# B&R Automation Studio project Parker_BMM_ST_V5_3147_V12 (part 22)

```c
				gPanelObj.idxKeyPicture[S$KEYMATRIX_F5] = STATE_SUB_PAGE;
					if(1 == EDGEPOS(gPanelObj.KeyMatric[S$KEYMATRIX_F5],KeyMatric[S$KEYMATRIX_F5]))
					{
					if(gPanelObj.PasswordLevel > 3)gPanelObj.SetPicture = PIC_OEM_SETTING_1;
				}
				if(gPanelObj.PasswordLevel <= 3)gPanelObj.idxKeyPicture[S$KEYMATRIX_F5] = STATE_INACTIVE;

					gPanelObj.idxKeyPicture[S$KEYMATRIX_F6] = STATE_SUB_PAGE;
					if(1 == EDGEPOS(gPanelObj.KeyMatric[S$KEYMATRIX_F6],KeyMatric[S$KEYMATRIX_F6]))
					{
					if(gPanelObj.PasswordLevel > 0)gPanelObj.SetPicture = PIC_PASSWORD_SET;
				}
				gPanelObj.idxKeyPicture[S$KEYMATRIX_F7] = STATE_SUB_PAGE;
					if(1 == EDGEPOS(gPanelObj.KeyMatric[S$KEYMATRIX_F7],KeyMatric[S$KEYMATRIX_F7]))
					{
					if(gPanelObj.PasswordLevel > 2)gPanelObj.SetPicture = PIC_PRESSURE_CALIBRATION ;
				}
				if(gPanelObj.PasswordLevel <= 2)gPanelObj.idxKeyPicture[S$KEYMATRIX_F7] = STATE_INACTIVE;
					//				gPanelObj.idxKeyPicture[S$KEYMATRIX_F7] = STATE_SUB_PAGE;
					//				if(1 == EDGEPOS(gPanelObj.KeyMatric[S$KEYMATRIX_F7],KeyMatric[S$KEYMATRIX_F7]))
					//				{
					//					if(0 == bLevel3CalibHide)
					//					{
					//						gPanelObj.SetPicture = PIC_MOLD_CALIBRATION;
					//					}
					//				}
					//				if(1 == bLevel3CalibHide)gPanelObj.idxKeyPicture[S$KEYMATRIX_F7] = STATE_INACTIVE;

					gPanelObj.idxKeyPicture[S$KEYMATRIX_F8] = STATE_SUB_PAGE;
					if(1 == EDGEPOS(gPanelObj.KeyMatric[S$KEYMATRIX_F8],KeyMatric[S$KEYMATRIX_F8]))
					{
					if(0 == bLevel3CalibHide)
					{
						if(ACTUATOR_ELECTRIC == gMachineFix.MoldR.Clamp.eActuatorType)
						{
							gPanelObj.SetPicture = PIC_CALIB_CLAMP_ENCODER;
						}
						else if(ACTUATOR_HYD == gMachineFix.MoldR.Clamp.eActuatorType )
						{
							gPanelObj.SetPicture = PIC_CALIB_CLAMP_LVDT;
						}

					}
				}
				if(1 == bLevel3CalibHide)gPanelObj.idxKeyPicture[S$KEYMATRIX_F8] = STATE_INACTIVE;

					//				gPanelObj.idxKeyPicture[S$KEYMATRIX_F7] = STATE_INACTIVE;
					//				gPanelObj.idxKeyPicture[S$KEYMATRIX_F8] = STATE_INACTIVE;

					gPanelObj.idxKeyPicture[S$KEYMATRIX_F9] = STATE_SUB_PAGE;
					if(1 == EDGEPOS(gPanelObj.KeyMatric[S$KEYMATRIX_F9],KeyMatric[S$KEYMATRIX_F9]))
					{
					if(gPanelObj.PasswordLevel > 3 && 1 == gTKcalib.Status)
					{
						gPanelObj.SetPicture = PIC_PROPORTION_VALVE;
					}
				}
				if(1 == bHidePropValvePage)gPanelObj.idxKeyPicture[S$KEYMATRIX_F9] = STATE_INACTIVE;

					gPanelObj.idxKeyPicture[S$KEYMATRIX_F10] = STATE_SUB_PAGE;
					if(1 == EDGEPOS(gPanelObj.KeyMatric[S$KEYMATRIX_F10],KeyMatric[S$KEYMATRIX_F10]))
					{
					gPanelObj.SetPicture = PIC_SCREEN_CALIBRATE;
				}

				gPanelObj.idxKeyPicture[S$KEYMATRIX_F11] = STATE_SUB_PAGE;
					if(1 == EDGEPOS(gPanelObj.KeyMatric[S$KEYMATRIX_F11],KeyMatric[S$KEYMATRIX_F11]))
					{
					if(gPanelObj.PasswordLevel > 2)gPanelObj.SetPicture = PIC_PV_LOG;
				}
				if(gPanelObj.PasswordLevel < 3)gPanelObj.idxKeyPicture[S$KEYMATRIX_F11] = STATE_INACTIVE;

					gPanelObj.idxKeyPicture[S$KEYMATRIX_F12] = STATE_SUB_PAGE;
					if(1 == EDGEPOS(gPanelObj.KeyMatric[S$KEYMATRIX_F12],KeyMatric[S$KEYMATRIX_F12]))
					{
					if(gPanelObj.PasswordLevel > 2)gPanelObj.SetPicture = PIC_LOG_INFO;
				}
				if(gPanelObj.PasswordLevel < 3)gPanelObj.idxKeyPicture[S$KEYMATRIX_F12] = STATE_INACTIVE;

					gPanelObj.idxKeyPicture[S$KEYMATRIX_F13] = STATE_SUB_PAGE;
					if(1 == EDGEPOS(gPanelObj.KeyMatric[S$KEYMATRIX_F13],KeyMatric[S$KEYMATRIX_F13]))
					{
					if(gPanelObj.PasswordLevel > 0)gPanelObj.SetPicture = PIC_INDUSTY_40;
				}
				if(gPanelObj.PasswordLevel < 1)gPanelObj.idxKeyPicture[S$KEYMATRIX_F13] = STATE_INACTIVE;

					gPanelObj.idxKeyPicture[S$KEYMATRIX_F14] = STATE_SUB_PAGE;
					if(1 == EDGEPOS(gPanelObj.KeyMatric[S$KEYMATRIX_F14],KeyMatric[S$KEYMATRIX_F14]))
					{
					if(gPanelObj.PasswordLevel > 0)gPanelObj.SetPicture = PIC_IP_CONFIG;
				}
				if(gPanelObj.PasswordLevel < 1)gPanelObj.idxKeyPicture[S$KEYMATRIX_F14] = STATE_INACTIVE;

					gPanelObj.idxKeyPicture[S$KEYMATRIX_F15] = STATE_SUB_PAGE;
					if(1 == EDGEPOS(gPanelObj.KeyMatric[S$KEYMATRIX_F15],KeyMatric[S$KEYMATRIX_F15]))
					{
					if(gPanelObj.PasswordLevel > 0)gPanelObj.SetPicture = PIC_VNC;
				}

				//						gPanelObj.idxKeyPicture[S$KEYMATRIX_F7] = STATE_INACTIVE;
				//            		gPanelObj.idxKeyPicture[S$KEYMATRIX_F8] = STATE_INACTIVE;
				//						gPanelObj.idxKeyPicture[S$KEYMATRIX_F8] = STATE_SUB_BUTTON;
				//						if(1 == EDGEPOS(gPanelObj.KeyMatric[S$KEYMATRIX_F8],KeyMatric[S$KEYMATRIX_F8]))
				//						{
				//						gMachineInfo.CycleTimes = 0;
				//						gCycleTimes             = 0;
				//						gMachineInfo.GoodBottles = 0;
				//					}

				//					gPanelObj.idxKeyPicture[S$KEYMATRIX_F9] = STATE_INACTIVE;
				//					gPanelObj.idxKeyPicture[S$KEYMATRIX_F10] = STATE_INACTIVE;
				//						gPanelObj.idxKeyPicture[S$KEYMATRIX_F10] = STATE_SUB_PAGE;
				//						if(1 == EDGEPOS(gPanelObj.KeyMatric[S$KEYMATRIX_F10],KeyMatric[S$KEYMATRIX_F10]))
				//						{
				//						gPanelObj.SetPicture = PIC_SCREEN_CALIBRATE;
				//					}
				//					gPanelObj.idxKeyPicture[S$KEYMATRIX_F11] = STATE_INACTIVE;
				//						gPanelObj.idxKeyPicture[S$KEYMATRIX_F12] = STATE_INACTIVE;
				//						gPanelObj.idxKeyPicture[S$KEYMATRIX_F13] = STATE_INACTIVE;
				//						gPanelObj.idxKeyPicture[S$KEYMATRIX_F14] = STATE_INACTIVE;
				//						gPanelObj.idxKeyPicture[S$KEYMATRIX_F15] = STATE_INACTIVE;

				gPanelObj.idxKeyPicture[S$KEYMATRIX_F16] = STATE_SUB_PAGE;
					if(1 == EDGEPOS(gPanelObj.KeyMatric[S$KEYMATRIX_F16],KeyMatric[S$KEYMATRIX_F16]))
					{
					gPanelObj.SetPicture = PIC_PASSWORD_LOGIN;
				}

				break;

			case PIC_PASSWORD_SET:
				//	case PIC_VALVE_DELAY:
			case PIC_PV_LOG:
				if(ChangePageDly > 0)
				{
					ChangePageDly--;
					break;
				}

				gPanelObj.idxKeyPicture[S$KEYMATRIX_F1] = STATE_SUB_PAGE;
				if(1 == EDGEPOS(gPanelObj.KeyMatric[S$KEYMATRIX_F1],KeyMatric[S$KEYMATRIX_F1]))
					{
					gPanelObj.SetPicture = PIC_OVERVIEW;
				}

				gPanelObj.idxKeyPicture[S$KEYMATRIX_F2] = STATE_SUB_PAGE;
					if(1 == EDGEPOS(gPanelObj.KeyMatric[S$KEYMATRIX_F2],KeyMatric[S$KEYMATRIX_F2]))
					{
					gPanelObj.SetPicture = gPanelObj.OldPicture;
				}

				gPanelObj.idxKeyPicture[S$KEYMATRIX_F3] = STATE_INACTIVE;
					gPanelObj.idxKeyPicture[S$KEYMATRIX_F4] = STATE_INACTIVE;
					gPanelObj.idxKeyPicture[S$KEYMATRIX_F5] = STATE_INACTIVE;

					gPanelObj.idxKeyPicture[S$KEYMATRIX_F6] = STATE_SUB_BUTTON;
					gPanelObj.idxKeyPicture[S$KEYMATRIX_F7] = STATE_SUB_BUTTON;

					gPanelObj.idxKeyPicture[S$KEYMATRIX_F8] = STATE_INACTIVE;
					gPanelObj.idxKeyPicture[S$KEYMATRIX_F9] = STATE_INACTIVE;
					gPanelObj.idxKeyPicture[S$KEYMATRIX_F10] = STATE_INACTIVE;
					gPanelObj.idxKeyPicture[S$KEYMATRIX_F11] = STATE_INACTIVE;
					gPanelObj.idxKeyPicture[S$KEYMATRIX_F12] = STATE_INACTIVE;
					gPanelObj.idxKeyPicture[S$KEYMATRIX_F13] = STATE_INACTIVE;
					gPanelObj.idxKeyPicture[S$KEYMATRIX_F14] = STATE_INACTIVE;
					gPanelObj.idxKeyPicture[S$KEYMATRIX_F15] = STATE_INACTIVE;
					gPanelObj.idxKeyPicture[S$KEYMATRIX_F16] = STATE_SUB_PAGE;
					if(1 == EDGEPOS(gPanelObj.KeyMatric[S$KEYMATRIX_F16],KeyMatric[S$KEYMATRIX_F16]))
					{
					gPanelObj.SetPicture = PIC_PASSWORD_LOGIN;
				}
				break;

			case PIC_SPC_CTRL:
			case PIC_SPC_1:
			case PIC_SPC_2:
				if(ChangePageDly > 0)
				{
					ChangePageDly--;
					break;
				}

				gPanelObj.idxKeyPicture[S$KEYMATRIX_F1] = STATE_SUB_PAGE;
					if(1 == EDGEPOS(gPanelObj.KeyMatric[S$KEYMATRIX_F1],KeyMatric[S$KEYMATRIX_F1]))
					{
					gPanelObj.SetPicture = PIC_OVERVIEW;
				}

				gPanelObj.idxKeyPicture[S$KEYMATRIX_F2] = STATE_SUB_PAGE;
					if(1 == EDGEPOS(gPanelObj.KeyMatric[S$KEYMATRIX_F2],KeyMatric[S$KEYMATRIX_F2]))
					{
					gPanelObj.SetPicture = gPanelObj.OldPicture;
				}

				gPanelObj.idxKeyPicture[S$KEYMATRIX_F3] = STATE_SUB_PAGE;
					if(1 == EDGEPOS(gPanelObj.KeyMatric[S$KEYMATRIX_F3],KeyMatric[S$KEYMATRIX_F3]))
					{
					gPanelObj.SetPicture = PIC_SPC_CTRL;
				}

				if(PIC_SPC_CTRL == gPanelObj.GetPicture)gPanelObj.idxKeyPicture[S$KEYMATRIX_F3]=STATE_ACTIVE;

					gPanelObj.idxKeyPicture[S$KEYMATRIX_F4] = STATE_SUB_PAGE;
					if(1 == EDGEPOS(gPanelObj.KeyMatric[S$KEYMATRIX_F4],KeyMatric[S$KEYMATRIX_F4]))
					{
					gPanelObj.SetPicture = PIC_SPC_1;
				}

				if(PIC_SPC_1 == gPanelObj.GetPicture)gPanelObj.idxKeyPicture[S$KEYMATRIX_F4]=STATE_ACTIVE;

					gPanelObj.idxKeyPicture[S$KEYMATRIX_F5] = STATE_SUB_PAGE;
					if(1 == EDGEPOS(gPanelObj.KeyMatric[S$KEYMATRIX_F5],KeyMatric[S$KEYMATRIX_F5]))
					{
					gPanelObj.SetPicture = PIC_SPC_2;
				}

				if(PIC_SPC_2 == gPanelObj.GetPicture)gPanelObj.idxKeyPicture[S$KEYMATRIX_F5]=STATE_ACTIVE;

					gPanelObj.idxKeyPicture[S$KEYMATRIX_F6] = STATE_INACTIVE;

					if(gPanelObj.GetPicture != PIC_SPC_CTRL)
				{
					gPanelObj.idxKeyPicture[S$KEYMATRIX_F7] = STATE_SUB_BUTTON;
						gPanelObj.idxKeyPicture[S$KEYMATRIX_F8] = STATE_SUB_BUTTON;
						}
				else
				{
					gPanelObj.idxKeyPicture[S$KEYMATRIX_F7] = STATE_INACTIVE;
						gPanelObj.idxKeyPicture[S$KEYMATRIX_F8] = STATE_INACTIVE;
						}

				gPanelObj.idxKeyPicture[S$KEYMATRIX_F9] = STATE_INACTIVE;
					gPanelObj.idxKeyPicture[S$KEYMATRIX_F10] = STATE_INACTIVE;
					gPanelObj.idxKeyPicture[S$KEYMATRIX_F11] = STATE_INACTIVE;
					gPanelObj.idxKeyPicture[S$KEYMATRIX_F12] = STATE_INACTIVE;
					gPanelObj.idxKeyPicture[S$KEYMATRIX_F13] = STATE_INACTIVE;
					gPanelObj.idxKeyPicture[S$KEYMATRIX_F14] = STATE_INACTIVE;
					gPanelObj.idxKeyPicture[S$KEYMATRIX_F15] = STATE_INACTIVE;
					gPanelObj.idxKeyPicture[S$KEYMATRIX_F16] = STATE_SUB_PAGE;
					if(1 == EDGEPOS(gPanelObj.KeyMatric[S$KEYMATRIX_F16],KeyMatric[S$KEYMATRIX_F16]))
					{
					gPanelObj.SetPicture = PIC_PASSWORD_LOGIN;
				}
				break;

			case PIC_HIGH_PASSWORD:
				if(ChangePageDly > 0)
				{
					ChangePageDly--;
					break;
				}

				gPanelObj.idxKeyPicture[S$KEYMATRIX_F1] = STATE_SUB_PAGE;
					if(1 == EDGEPOS(gPanelObj.KeyMatric[S$KEYMATRIX_F1],KeyMatric[S$KEYMATRIX_F1]))
					{
					gPanelObj.SetPicture = PIC_OVERVIEW;
				}

				gPanelObj.idxKeyPicture[S$KEYMATRIX_F2] = STATE_SUB_PAGE;
					if(1 == EDGEPOS(gPanelObj.KeyMatric[S$KEYMATRIX_F2],KeyMatric[S$KEYMATRIX_F2]))
					{
					gPanelObj.SetPicture = gPanelObj.OldPicture;
				}

				gPanelObj.idxKeyPicture[S$KEYMATRIX_F3] = STATE_INACTIVE;

					gPanelObj.idxKeyPicture[S$KEYMATRIX_F4] = STATE_INACTIVE;
					if(1 == EDGEPOS(gPanelObj.KeyMatric[S$KEYMATRIX_F4],KeyMatric[S$KEYMATRIX_F4]))
					{
					if(PIC_HIGH_PASSWORD == gPanelObj.GetPicture)
					{
						gPwd.Option[0] = !gPwd.Option[0];
						gPwd.wSavePassword = 1;
					}
				}
				if(gPanelObj.GetPicture == PIC_HIGH_PASSWORD)gPanelObj.idxKeyPicture[S$KEYMATRIX_F4] = STATE_SUB_BUTTON;

					gPanelObj.idxKeyPicture[S$KEYMATRIX_F5] = STATE_INACTIVE;
					if(1 == EDGEPOS(gPanelObj.KeyMatric[S$KEYMATRIX_F5],KeyMatric[S$KEYMATRIX_F5]))
					{
					if(PIC_HIGH_PASSWORD == gPanelObj.GetPicture)
					{
						gPwd.Option[1] = !gPwd.Option[1];
						gPwd.wSavePassword = 1;
					}
				}
				if(gPanelObj.GetPicture == PIC_HIGH_PASSWORD)gPanelObj.idxKeyPicture[S$KEYMATRIX_F5] = STATE_SUB_BUTTON;

					gPanelObj.idxKeyPicture[S$KEYMATRIX_F6] = STATE_INACTIVE;
					if(1 == EDGEPOS(gPanelObj.KeyMatric[S$KEYMATRIX_F6],KeyMatric[S$KEYMATRIX_F6]))
					{
					if(PIC_HIGH_PASSWORD == gPanelObj.GetPicture)
					{
						gPwd.Option[2] = !gPwd.Option[2];
						gPwd.wSavePassword = 1;
					}
				}
				if(gPanelObj.GetPicture == PIC_HIGH_PASSWORD)gPanelObj.idxKeyPicture[S$KEYMATRIX_F6] = STATE_SUB_BUTTON;

					gPanelObj.idxKeyPicture[S$KEYMATRIX_F7] = STATE_INACTIVE;

					gPanelObj.idxKeyPicture[S$KEYMATRIX_F8] = STATE_INACTIVE;
					if(1 == EDGEPOS(gPanelObj.KeyMatric[S$KEYMATRIX_F8],KeyMatric[S$KEYMATRIX_F8]))
					{
					if(PIC_HIGH_PASSWORD == gPanelObj.GetPicture)
					{
						gMachineStopDays = 0;

						gPwd.OK_3 = 0;
						gPwd.OK_2 = 0;
						gPwd.OK_1 = 0;

						gPwd.wSavePassword = 1;
					}
				}
				if(gPanelObj.GetPicture == PIC_HIGH_PASSWORD)gPanelObj.idxKeyPicture[S$KEYMATRIX_F8] = STATE_SUB_BUTTON;

					gPanelObj.idxKeyPicture[S$KEYMATRIX_F9] = STATE_INACTIVE;
					gPanelObj.idxKeyPicture[S$KEYMATRIX_F10] = STATE_INACTIVE;
					gPanelObj.idxKeyPicture[S$KEYMATRIX_F11] = STATE_INACTIVE;
					gPanelObj.idxKeyPicture[S$KEYMATRIX_F12] = STATE_INACTIVE;
					gPanelObj.idxKeyPicture[S$KEYMATRIX_F13] = STATE_INACTIVE;
					if(gPanelObj.GetPicture == PIC_INDUSTY_40)gPanelObj.idxKeyPicture[S$KEYMATRIX_F13] = STATE_ACTIVE;
					gPanelObj.idxKeyPicture[S$KEYMATRIX_F14] = STATE_INACTIVE;
					gPanelObj.idxKeyPicture[S$KEYMATRIX_F15] = STATE_INACTIVE;
					gPanelObj.idxKeyPicture[S$KEYMATRIX_F16] = STATE_SUB_PAGE;
					if(1 == EDGEPOS(gPanelObj.KeyMatric[S$KEYMATRIX_F16],KeyMatric[S$KEYMATRIX_F16]))
					{
					gPanelObj.SetPicture = PIC_PASSWORD_LOGIN;
				}
				break;

			case PIC_INIT_SET:
				if(ChangePageDly > 0)
				{
					ChangePageDly--;
					break;
				}

				gPanelObj.idxKeyPicture[S$KEYMATRIX_F1] = STATE_SUB_PAGE;
					if(1 == EDGEPOS(gPanelObj.KeyMatric[S$KEYMATRIX_F1],KeyMatric[S$KEYMATRIX_F1]))
					{
					gPanelObj.SetPicture = PIC_OVERVIEW;
				}

				gPanelObj.idxKeyPicture[S$KEYMATRIX_F2] = STATE_SUB_PAGE;
					if(1 == EDGEPOS(gPanelObj.KeyMatric[S$KEYMATRIX_F2],KeyMatric[S$KEYMATRIX_F2]))
					{
					gPanelObj.SetPicture = gPanelObj.OldPicture;
				}

				gPanelObj.idxKeyPicture[S$KEYMATRIX_F3] = STATE_ACTIVE;
					if(1 == EDGEPOS(gPanelObj.KeyMatric[S$KEYMATRIX_F3],KeyMatric[S$KEYMATRIX_F3]))
					{
					gPanelObj.SetPicture = PIC_THICK_START;
				}
				gPanelObj.idxKeyPicture[S$KEYMATRIX_F4] = STATE_INACTIVE;
					gPanelObj.idxKeyPicture[S$KEYMATRIX_F5] = STATE_INACTIVE;
					gPanelObj.idxKeyPicture[S$KEYMATRIX_F6] = STATE_INACTIVE;
					gPanelObj.idxKeyPicture[S$KEYMATRIX_F7] = STATE_INACTIVE;
					gPanelObj.idxKeyPicture[S$KEYMATRIX_F8] = STATE_INACTIVE;
					gPanelObj.idxKeyPicture[S$KEYMATRIX_F9] = STATE_INACTIVE;
					gPanelObj.idxKeyPicture[S$KEYMATRIX_F10] = STATE_INACTIVE;
					gPanelObj.idxKeyPicture[S$KEYMATRIX_F11] = STATE_INACTIVE;

					if(1 == EDGEPOS(gPanelObj.KeyMatric[S$KEYMATRIX_F12],KeyMatric[S$KEYMATRIX_F12]))
					{
					gPanelObj.SetPicture = PIC_THICK_DIVER;
				}
				//					gPanelObj.idxKeyPicture[S$KEYMATRIX_F6] = STATE_SUB_BUTTON;
				//					if(1 == EDGEPOS(gPanelObj.KeyMatric[S$KEYMATRIX_F6],KeyMatric[S$KEYMATRIX_F6]))
				//					{
				//					gThickProf.FunOption.bLengthUnit = !gThickProf.FunOption.bLengthUnit;
				//					gRecipeOperate.OnceSave = 1;
				//				}
				//
				//				gPanelObj.idxKeyPicture[S$KEYMATRIX_F7] = STATE_SUB_BUTTON;
				//					if(1 == EDGEPOS(gPanelObj.KeyMatric[S$KEYMATRIX_F7],KeyMatric[S$KEYMATRIX_F7]))
				//					{
				//					gThickProf.FunOption.IsTraceInEdit = !gThickProf.FunOption.IsTraceInEdit;
				//					gRecipeOperate.OnceSave = 1;
				//				}
				//
				//				gPanelObj.idxKeyPicture[S$KEYMATRIX_F8] = STATE_SUB_BUTTON;
				//					if(1 == EDGEPOS(gPanelObj.KeyMatric[S$KEYMATRIX_F8],KeyMatric[S$KEYMATRIX_F8]))
				//					{
				//					gThickProf.FunOption.Is100_300 = !gThickProf.FunOption.Is100_300;
				//					gRecipeOperate.OnceSave = 1;
				//				}
				//
				//				gPanelObj.idxKeyPicture[S$KEYMATRIX_F9] = STATE_SUB_BUTTON;
				//					if(1 == EDGEPOS(gPanelObj.KeyMatric[S$KEYMATRIX_F9],KeyMatric[S$KEYMATRIX_F9]))
				//					{
				//					gThickProf.FunOption.IsZeroDn = !gThickProf.FunOption.IsZeroDn;
				//					gRecipeOperate.OnceSave = 1;
				//				}
				//
				//				gPanelObj.idxKeyPicture[S$KEYMATRIX_F10] = STATE_SUB_BUTTON;
				//					if(1 == EDGEPOS(gPanelObj.KeyMatric[S$KEYMATRIX_F10],KeyMatric[S$KEYMATRIX_F10]))
				//					{
				//					gThickProf.FunOption.SealMode = !gThickProf.FunOption.SealMode;
				//					gRecipeOperate.OnceSave = 1;
				//				}
				//
				//				gPanelObj.idxKeyPicture[S$KEYMATRIX_F11] = STATE_INACTIVE;
				//
				//					gPanelObj.idxKeyPicture[S$KEYMATRIX_F12] = STATE_SUB_BUTTON;
				//					if(1 == EDGEPOS(gPanelObj.KeyMatric[S$KEYMATRIX_F12],KeyMatric[S$KEYMATRIX_F12]))
				//					{
				//					gThickProf.FunOption.Servo = !gThickProf.FunOption.Servo;
				//					gRecipeOperate.OnceSave = 1;
				//				}

				gPanelObj.idxKeyPicture[S$KEYMATRIX_F13] = STATE_SUB_PAGE;
					if(1 == EDGENEG(gPanelObj.KeyMatric[S$KEYMATRIX_F13],KeyMatric[S$KEYMATRIX_F13]))
					{
					//	if(gPanelObj.PasswordLevel > 2 &&  1 == gTKcalib.Status)
					if(gPanelObj.PasswordLevel > 2 &&  0 == gTKauto.Status)

					{
						gPanelObj.SetPicture = PIC_INIT_SET  ;
						OldSet    = gThickProf.ShareSet;
						OldFunSet = gThickProf.FunOption;
					}
				}
				//	if(1 == bThickCalibHide)gPanelObj.idxKeyPicture[S$KEYMATRIX_F13] = STATE_INACTIVE;
				if(1 == gTKauto.Status)gPanelObj.idxKeyPicture[S$KEYMATRIX_F13] = STATE_INACTIVE;

					gPanelObj.idxKeyPicture[S$KEYMATRIX_F14] = STATE_SUB_PAGE;
					if(1 == EDGENEG(gPanelObj.KeyMatric[S$KEYMATRIX_F14],KeyMatric[S$KEYMATRIX_F14]))
					{
					//	if(gPanelObj.PasswordLevel > 2 &&  1 == gTKcalib.Status)
					if(gPanelObj.PasswordLevel > 2 &&  0 == gTKauto.Status)
					{
						gPanelObj.SetPicture = PIC_GAP_CALIBRATE;
						OldSet    = gThickProf.ShareSet;
						OldFunSet = gThickProf.FunOption;
					}
				}
				//if(1 == bThickCalibHide)gPanelObj.idxKeyPicture[S$KEYMATRIX_F14] = STATE_INACTIVE;
				if(1 == gTKauto.Status)gPanelObj.idxKeyPicture[S$KEYMATRIX_F14] = STATE_INACTIVE;
					gPanelObj.idxKeyPicture[S$KEYMATRIX_F15] = STATE_INACTIVE;
					gPanelObj.idxKeyPicture[S$KEYMATRIX_F16] = STATE_SUB_PAGE;
					if(1 == EDGEPOS(gPanelObj.KeyMatric[S$KEYMATRIX_F16],KeyMatric[S$KEYMATRIX_F16]))
					{
					gPanelObj.SetPicture = PIC_PASSWORD_LOGIN;
				}

				if(gThickProf.ShareSet.StartFlow > 998)gThickProf.ShareSet.StartFlow = 998;
				if(gThickProf.ShareSet.SealFlow  > 998)gThickProf.ShareSet.SealFlow  = 998;
				if(gThickProf.ShareSet.ThickFlow > 998)gThickProf.ShareSet.ThickFlow = 998;

				if(gThickProf.ShareSet.StartFlow < 100)gThickProf.ShareSet.StartFlow = 100;
				if(gThickProf.ShareSet.SealFlow  < 100)gThickProf.ShareSet.SealFlow  = 100;
				if(gThickProf.ShareSet.ThickFlow < 100)gThickProf.ShareSet.ThickFlow = 100;
				break;

			case PIC_GAP_CALIBRATE:
				if(ChangePageDly > 0)
				{
					ChangePageDly--;
					break;
				}

				gPanelObj.idxKeyPicture[S$KEYMATRIX_F1] = STATE_SUB_PAGE;
					if(1 == EDGEPOS(gPanelObj.KeyMatric[S$KEYMATRIX_F1],KeyMatric[S$KEYMATRIX_F1]))
					{
					gPanelObj.SetPicture = PIC_OVERVIEW;
				}

				gPanelObj.idxKeyPicture[S$KEYMATRIX_F2] = STATE_SUB_PAGE;
					if(1 == EDGEPOS(gPanelObj.KeyMatric[S$KEYMATRIX_F2],KeyMatric[S$KEYMATRIX_F2]))
					{
					gPanelObj.SetPicture = gPanelObj.OldPicture;
				}

				gPanelObj.idxKeyPicture[S$KEYMATRIX_F3] = STATE_ACTIVE;
					if(1 == EDGEPOS(gPanelObj.KeyMatric[S$KEYMATRIX_F3],KeyMatric[S$KEYMATRIX_F3]))
					{
					gPanelObj.SetPicture = PIC_THICK_START;
				}
				gPanelObj.idxKeyPicture[S$KEYMATRIX_F4]  = STATE_INACTIVE;

					if(gMachineFix.Parison.eActuatorType == ACTUATOR_ELECTRIC)
				{
					//Electric

					if (gPanelObj.GetPicture ==PIC_GAP_CALIBRATE )
					{
						gPanelObj.idxKeyPicture[S$KEYMATRIX_F5] = STATE_SUB_BUTTON;
							if(1 == EDGEPOS(gPanelObj.KeyMatric[S$KEYMATRIX_F5],KeyMatric[S$KEYMATRIX_F5]))
							{
							if(1 == gMachineInfo.Calib)
							{
								gThickIO.Step = STEP_THICK_CALIB_DOWN;
							}
						}

						if(1 == EDGENEG(gPanelObj.KeyMatric[S$KEYMATRIX_F5],keyF5N))
							{
							if(1 == gMachineInfo.Calib)
							{
								gThickIO.Step = STEP_THICK_STOP;
							}
						}

						gPanelObj.idxKeyPicture[S$KEYMATRIX_F6] = STATE_SUB_BUTTON;
							if(1 == EDGEPOS(gPanelObj.KeyMatric[S$KEYMATRIX_F6],KeyMatric[S$KEYMATRIX_F6]))
							{
							if(1 == gMachineInfo.Calib)
							{
								gThickIO.Step = STEP_THICK_CALIB_UP;
							}
						}

						if(1 == EDGENEG(gPanelObj.KeyMatric[S$KEYMATRIX_F6],keyF6N))
							{
							if(1 == gMachineInfo.Calib)
							{
								gThickIO.Step = STEP_THICK_STOP;
							}
						}
						gPanelObj.idxKeyPicture[S$KEYMATRIX_F7] = STATE_SUB_BUTTON;
							if(1 == EDGEPOS(gPanelObj.KeyMatric[S$KEYMATRIX_F7],KeyMatric[S$KEYMATRIX_F7]))
							{
							if(1 == gMachineInfo.Calib)
							{
								gThickFix.ecMin = gThickIO.ecAs;
								gRecipeOperate.OnceSave = 1;
							}
						}

						gPanelObj.idxKeyPicture[S$KEYMATRIX_F8] = STATE_SUB_BUTTON;
							if(1 == EDGEPOS(gPanelObj.KeyMatric[S$KEYMATRIX_F8],KeyMatric[S$KEYMATRIX_F8]))
							{
							if(1 == gMachineInfo.Calib)
							{
								gThickFix.ecMax = gThickIO.ecAs;
								gRecipeOperate.OnceSave = 1;
							}
						}
					}

					gPanelObj.idxKeyPicture[S$KEYMATRIX_F9]  = STATE_INACTIVE;
						gPanelObj.idxKeyPicture[S$KEYMATRIX_F10] = STATE_INACTIVE;
						gPanelObj.idxKeyPicture[S$KEYMATRIX_F11] = STATE_INACTIVE;

						gPanelObj.idxKeyPicture[S$KEYMATRIX_F12] = STATE_SUB_PAGE;
						if(1 == EDGEPOS(gPanelObj.KeyMatric[S$KEYMATRIX_F12],KeyMatric[S$KEYMATRIX_F12]))
						{
						gPanelObj.SetPicture = PIC_THICK_DIVER;
					}

				}
				else if(gMachineFix.Parison.eActuatorType == ACTUATOR_HYD)
				{
					//Hydraulic

					gPanelObj.idxKeyPicture[S$KEYMATRIX_F5] = STATE_SUB_BUTTON;
						gPanelObj.idxKeyPicture[S$KEYMATRIX_F6] = STATE_SUB_BUTTON;
						gPanelObj.idxKeyPicture[S$KEYMATRIX_F7] = STATE_SUB_BUTTON;
						if(1 == gPanelObj.KeyMatric[S$KEYMATRIX_F7])
						{
						cntF7 = cntF7 + 1;
					}
					else
					{
						cntF7 = 0;
					}
					if(50 == cntF7)
					{
						if(gServoLinear.Current > 0 && gServoLinear.Current < 32767)
						{
							gServoLinear.ZeroPos     = gServoLinear.Current;
							gRecipeOperate.OnceSave = 1;
						}
					}

					gPanelObj.idxKeyPicture[S$KEYMATRIX_F8] = STATE_SUB_BUTTON;
						if(1 == gPanelObj.KeyMatric[S$KEYMATRIX_F8])
						{
						cntF8 = cntF8 + 1;
					}
					else
					{
						cntF8 = 0;
					}

					if(50 == cntF8)
					{
						if(gServoLinear.Current > 0 && gServoLinear.Current < 32767)
						{
							if(gServoLinear.Current > gServoLinear.ZeroPos)
							{
								gServoLinear.MaxPos      = gServoLinear.Current;
								gRecipeOperate.OnceSave = 1;
							}
						}
					}

					// auto calibration
					if(1 == gThickProf.FunOption.IsAutoCalibrate)
					{
						gPanelObj.idxKeyPicture[S$KEYMATRIX_F11] = STATE_SUB_BUTTON;
							bHideParisonAutoCalib = 0;

						if(1 == gPanelObj.KeyMatric[S$KEYMATRIX_F5] || 1 == gPanelObj.KeyMatric[S$KEYMATRIX_F6] ||
							1 == gPanelObj.KeyMatric[S$KEYMATRIX_F7] || 1 == gPanelObj.KeyMatric[S$KEYMATRIX_F8])
							{
							gImply.ParisonCalibNotManual = 1;
						}
					}
					else
					{
						gPanelObj.idxKeyPicture[S$KEYMATRIX_F11] = STATE_INACTIVE;
							bHideParisonAutoCalib = 1;
					}

					gPanelObj.idxKeyPicture[S$KEYMATRIX_F9]  = STATE_INACTIVE;
						gPanelObj.idxKeyPicture[S$KEYMATRIX_F10] = STATE_INACTIVE;

						gPanelObj.idxKeyPicture[S$KEYMATRIX_F12] = STATE_INACTIVE;

						}

				/*-------------------F13----------------------*/
				gPanelObj.idxKeyPicture[S$KEYMATRIX_F13] = STATE_SUB_PAGE;
					if(1 == EDGENEG(gPanelObj.KeyMatric[S$KEYMATRIX_F13],KeyMatric[S$KEYMATRIX_F13]))
					{
					//	if(gPanelObj.PasswordLevel > 2 &&  1 == gTKcalib.Status)
					if(gPanelObj.PasswordLevel > 2 &&  0 == gTKauto.Status)

					{
						gPanelObj.SetPicture = PIC_INIT_SET  ;
						OldSet    = gThickProf.ShareSet;
						OldFunSet = gThickProf.FunOption;
					}
				}

				if(1 == gTKauto.Status)gPanelObj.idxKeyPicture[S$KEYMATRIX_F13] = STATE_INACTIVE;

					/*-------------------F14----------------------*/
					gPanelObj.idxKeyPicture[S$KEYMATRIX_F14] = STATE_SUB_PAGE;
					if(1 == EDGENEG(gPanelObj.KeyMatric[S$KEYMATRIX_F14],KeyMatric[S$KEYMATRIX_F14]))
					{
					//	if(gPanelObj.PasswordLevel > 2 &&  1 == gTKcalib.Status)
					if(gPanelObj.PasswordLevel > 2 &&  0 == gTKauto.Status)
					{
						gPanelObj.SetPicture = PIC_GAP_CALIBRATE;
						OldSet    = gThickProf.ShareSet;
						OldFunSet = gThickProf.FunOption;
					}
				}
				//if(1 == bThickCalibHide)gPanelObj.idxKeyPicture[S$KEYMATRIX_F14] = STATE_INACTIVE;
				if(1 == gTKauto.Status)gPanelObj.idxKeyPicture[S$KEYMATRIX_F14] = STATE_INACTIVE;
					if(1 == EDGEPOS(gPanelObj.KeyMatric[S$KEYMATRIX_F15],KeyMatric[S$KEYMATRIX_F15]))
					{
					gPanelObj.SetPicture = PIC_GAP_CALIBRATE_HELP;
				}
				gPanelObj.idxKeyPicture[S$KEYMATRIX_F16] = STATE_SUB_PAGE;
					if(1 == EDGEPOS(gPanelObj.KeyMatric[S$KEYMATRIX_F16],KeyMatric[S$KEYMATRIX_F16]))
					{
					gPanelObj.SetPicture = PIC_PASSWORD_LOGIN;
				}
				break;

			case PIC_GAP_CALIBRATE_HELP:
				if(ChangePageDly > 0)
				{
					ChangePageDly--;
					break;
				}

				gPanelObj.idxKeyPicture[S$KEYMATRIX_F1] = STATE_SUB_PAGE;
					if(1 == EDGEPOS(gPanelObj.KeyMatric[S$KEYMATRIX_F1],KeyMatric[S$KEYMATRIX_F1]))
					{
					gPanelObj.SetPicture = PIC_GAP_CALIBRATE;
				}

				gPanelObj.idxKeyPicture[S$KEYMATRIX_F2] = STATE_INACTIVE;
					gPanelObj.idxKeyPicture[S$KEYMATRIX_F3] = STATE_INACTIVE;
					gPanelObj.idxKeyPicture[S$KEYMATRIX_F4] = STATE_INACTIVE;
					gPanelObj.idxKeyPicture[S$KEYMATRIX_F5] = STATE_INACTIVE;
					gPanelObj.idxKeyPicture[S$KEYMATRIX_F6] = STATE_INACTIVE;
					gPanelObj.idxKeyPicture[S$KEYMATRIX_F7] = STATE_INACTIVE;
					gPanelObj.idxKeyPicture[S$KEYMATRIX_F8] = STATE_INACTIVE;
					gPanelObj.idxKeyPicture[S$KEYMATRIX_F9] = STATE_INACTIVE;
					gPanelObj.idxKeyPicture[S$KEYMATRIX_F10] = STATE_INACTIVE;
					gPanelObj.idxKeyPicture[S$KEYMATRIX_F11] = STATE_INACTIVE;
					gPanelObj.idxKeyPicture[S$KEYMATRIX_F12] = STATE_INACTIVE;
					gPanelObj.idxKeyPicture[S$KEYMATRIX_F13] = STATE_INACTIVE;
					gPanelObj.idxKeyPicture[S$KEYMATRIX_F14] = STATE_INACTIVE;
					gPanelObj.idxKeyPicture[S$KEYMATRIX_F15] = STATE_INACTIVE;
					gPanelObj.idxKeyPicture[S$KEYMATRIX_F16] = STATE_SUB_PAGE;
					if(1 == EDGEPOS(gPanelObj.KeyMatric[S$KEYMATRIX_F16],KeyMatric[S$KEYMATRIX_F16]))
					{
					gPanelObj.SetPicture = PIC_PASSWORD_LOGIN;
				}
				break;

			case PIC_DEFAULT_SET:
				if(ChangePageDly > 0)
				{
					ChangePageDly--;
					break;
				}

				gPanelObj.idxKeyPicture[S$KEYMATRIX_F1] = STATE_SUB_PAGE;
					if(1 == EDGEPOS(gPanelObj.KeyMatric[S$KEYMATRIX_F1],KeyMatric[S$KEYMATRIX_F1]))
					{
					gPanelObj.SetPicture = PIC_OVERVIEW;
				}

				gPanelObj.idxKeyPicture[S$KEYMATRIX_F2] = STATE_SUB_PAGE;
					if(1 == EDGEPOS(gPanelObj.KeyMatric[S$KEYMATRIX_F2],KeyMatric[S$KEYMATRIX_F2]))
					{
					gPanelObj.SetPicture = gPanelObj.OldPicture;
				}

				gPanelObj.idxKeyPicture[S$KEYMATRIX_F3] = STATE_SUB_PAGE;
					if(1 == EDGEPOS(gPanelObj.KeyMatric[S$KEYMATRIX_F3],KeyMatric[S$KEYMATRIX_F3]))
					{
					gPanelObj.SetPicture = PIC_GAP_CALIBRATE;
				}

				gPanelObj.idxKeyPicture[S$KEYMATRIX_F4] = STATE_INACTIVE;
					gPanelObj.idxKeyPicture[S$KEYMATRIX_F5] = STATE_INACTIVE;
					gPanelObj.idxKeyPicture[S$KEYMATRIX_F6] = STATE_INACTIVE;
					gPanelObj.idxKeyPicture[S$KEYMATRIX_F7] = STATE_INACTIVE;
					gPanelObj.idxKeyPicture[S$KEYMATRIX_F8] = STATE_INACTIVE;
					gPanelObj.idxKeyPicture[S$KEYMATRIX_F9] = STATE_INACTIVE;

					gPanelObj.idxKeyPicture[S$KEYMATRIX_F10] = STATE_INACTIVE;
					gPanelObj.idxKeyPicture[S$KEYMATRIX_F11] = STATE_INACTIVE;
					gPanelObj.idxKeyPicture[S$KEYMATRIX_F12] = STATE_INACTIVE;
					gPanelObj.idxKeyPicture[S$KEYMATRIX_F13] = STATE_INACTIVE;
					gPanelObj.idxKeyPicture[S$KEYMATRIX_F14] = STATE_INACTIVE;
					gPanelObj.idxKeyPicture[S$KEYMATRIX_F15] = STATE_INACTIVE;
					gPanelObj.idxKeyPicture[S$KEYMATRIX_F16] = STATE_SUB_PAGE;
					if(1 == EDGEPOS(gPanelObj.KeyMatric[S$KEYMATRIX_F16],KeyMatric[S$KEYMATRIX_F16]))
					{
					gPanelObj.SetPicture = PIC_PASSWORD_LOGIN;
				}
				break;

			case PIC_CALIB_CLAMP_ENCODER:
			case PIC_CALIB_CARRIAGE_ENCODER:
			case PIC_CALIB_BLOWPIN_ENCODER:
			case PIC_CALIB_OTHER_ENCODER:
			case PIC_CALIB_ROBOT_ENCODER:
			case PIC_CALIB_CLAMP_LVDT:
			case PIC_CALIB_CARRIAGE_LVDT:
			case PIC_CALIB_BLOWPIN_LVDT:

				if(ChangePageDly > 0)
				{
					ChangePageDly--;
					break;
				}

				gPanelObj.idxKeyPicture[S$KEYMATRIX_F1] = STATE_SUB_PAGE;
					if(1 == EDGEPOS(gPanelObj.KeyMatric[S$KEYMATRIX_F1],KeyMatric[S$KEYMATRIX_F1]))
					{
					gPanelObj.SetPicture = PIC_OVERVIEW;
				}

				gPanelObj.idxKeyPicture[S$KEYMATRIX_F2] = STATE_SUB_PAGE;
					if(1 == EDGEPOS(gPanelObj.KeyMatric[S$KEYMATRIX_F2],KeyMatric[S$KEYMATRIX_F2]))
					{
					gPanelObj.SetPicture = gPanelObj.OldPicture;
				}

				gPanelObj.idxKeyPicture[S$KEYMATRIX_F3] = STATE_SUB_PAGE;
					if(1 == EDGEPOS(gPanelObj.KeyMatric[S$KEYMATRIX_F3],KeyMatric[S$KEYMATRIX_F3]))
					{
					gPanelObj.SetPicture = PIC_CALIB_CLAMP_ENCODER;
				}
				if( 1 == bHideClampActuatorElectic )gPanelObj.idxKeyPicture[S$KEYMATRIX_F3] = STATE_INACTIVE;

					gPanelObj.idxKeyPicture[S$KEYMATRIX_F4] = STATE_SUB_PAGE;
					if(1 == EDGEPOS(gPanelObj.KeyMatric[S$KEYMATRIX_F4],KeyMatric[S$KEYMATRIX_F4]))
					{
					gPanelObj.SetPicture = PIC_CALIB_CARRIAGE_ENCODER;

				}
				if( 1 == bHideCarriageActuatorElectic )gPanelObj.idxKeyPicture[S$KEYMATRIX_F4] = STATE_INACTIVE;

					gPanelObj.idxKeyPicture[S$KEYMATRIX_F5] = STATE_SUB_PAGE;
					if(1 == EDGEPOS(gPanelObj.KeyMatric[S$KEYMATRIX_F5],KeyMatric[S$KEYMATRIX_F5]))
					{
					gPanelObj.SetPicture = PIC_CALIB_BLOWPIN_ENCODER;
				}
				if( 1 == bHideBlowPinActuatorElectic)gPanelObj.idxKeyPicture[S$KEYMATRIX_F5] = STATE_INACTIVE;

					gPanelObj.idxKeyPicture[S$KEYMATRIX_F6] = STATE_SUB_PAGE;
					if(1 == EDGEPOS(gPanelObj.KeyMatric[S$KEYMATRIX_F6],KeyMatric[S$KEYMATRIX_F6]))
					{
					if( 0 == bHideClampActuatorHyd_LVDT)gPanelObj.SetPicture = PIC_CALIB_CLAMP_LVDT;
				}
				if( 1 == bHideClampActuatorHyd_LVDT)gPanelObj.idxKeyPicture[S$KEYMATRIX_F6] = STATE_INACTIVE;

					gPanelObj.idxKeyPicture[S$KEYMATRIX_F7] = STATE_SUB_PAGE;
					if(1 == EDGEPOS(gPanelObj.KeyMatric[S$KEYMATRIX_F7],KeyMatric[S$KEYMATRIX_F7]))
					{
					if( 0 == bHideCarriageActuatorHyd_LVDT)gPanelObj.SetPicture = PIC_CALIB_CARRIAGE_LVDT;
				}
				if( 1 == bHideCarriageActuatorHyd_LVDT)gPanelObj.idxKeyPicture[S$KEYMATRIX_F7] = STATE_INACTIVE;

					gPanelObj.idxKeyPicture[S$KEYMATRIX_F8] = STATE_SUB_PAGE;
					if(1 == EDGEPOS(gPanelObj.KeyMatric[S$KEYMATRIX_F8],KeyMatric[S$KEYMATRIX_F8]))
					{
					if( 0 == bHideBlowPinActuatorHyd_LVDT)gPanelObj.SetPicture = PIC_CALIB_BLOWPIN_LVDT;
				}
				if( 1 == bHideBlowPinActuatorHyd_LVDT)gPanelObj.idxKeyPicture[S$KEYMATRIX_F8] = STATE_INACTIVE;

					gPanelObj.idxKeyPicture[S$KEYMATRIX_F9] = STATE_SUB_PAGE;
					if(1 == EDGEPOS(gPanelObj.KeyMatric[S$KEYMATRIX_F9],KeyMatric[S$KEYMATRIX_F9]))
					{
					gPanelObj.SetPicture = PIC_CALIB_OTHER_ENCODER;
				}
				if( 1 == bHideExtrLiftActuatorElectric)gPanelObj.idxKeyPicture[S$KEYMATRIX_F9] = STATE_INACTIVE;

					gPanelObj.idxKeyPicture[S$KEYMATRIX_F10] = STATE_SUB_PAGE;
					if(1 == EDGEPOS(gPanelObj.KeyMatric[S$KEYMATRIX_F10],KeyMatric[S$KEYMATRIX_F10]))
					{
					gPanelObj.SetPicture = PIC_CALIB_ROBOT_ENCODER;
				}
				if( 1 == bHideRobotTransferActuatorElec)gPanelObj.idxKeyPicture[S$KEYMATRIX_F10] = STATE_INACTIVE;

					gPanelObj.idxKeyPicture[S$KEYMATRIX_F11] = STATE_INACTIVE;
					gPanelObj.idxKeyPicture[S$KEYMATRIX_F12] = STATE_INACTIVE;

					/*----Reset Calibrate Function---------*/
					/* check commands */
					if (((bCmdResetClampR) || (bCmdResetClampL) || (bCmdResetBlowPinR) || (bCmdResetBlowPinL) || (bCmdResetCarriageR) || (bCmdResetCarriageL)|| (bCmdResetBlowPin2R) || (bCmdResetBlowPin2L) || (bCmdResetExtrLift) )&& (gPanelObj.PasswordLevel > 3))
				{
					uHideDiagResetCalib = 0;
				}

				/*Dialog Pop up contorl*/

				if(0 == uHideDiagResetCalib)
				{
					if(bConfirmReset)
					{
						if(bCmdResetClampR)
						{
							gMachineFix.MoldR.Clamp.Zero = 0;
							gMachineFix.MoldR.Clamp.Max = 0;
							gRecipeOperate.OnceSave = 1;
							bCmdResetClampR = 0;
						}
						else if(bCmdResetClampL)
						{
							gMachineFix.MoldL.Clamp.Zero = 0;
							gMachineFix.MoldL.Clamp.Max = 0;
							gRecipeOperate.OnceSave = 1;
							bCmdResetClampL = 0;
						}
						else if(bCmdResetBlowPinR)
						{
							gMachineFix.MoldR.BlowPin.Zero = 0;
							gMachineFix.MoldR.BlowPin.Max = 0;
							gRecipeOperate.OnceSave = 1;
							bCmdResetBlowPinR = 0;
						}
						else if(bCmdResetBlowPinL)
						{
							gMachineFix.MoldL.BlowPin.Zero = 0;
							gMachineFix.MoldL.BlowPin.Max = 0;
							gRecipeOperate.OnceSave = 1;
							bCmdResetBlowPinL = 0;
						}
						else if(bCmdResetCarriageR)
						{
							gMachineFix.MoldR.Carriage.Zero = 0;
							gMachineFix.MoldR.Carriage.Max = 0;
							gRecipeOperate.OnceSave = 1;
							bCmdResetCarriageR = 0;
						}
						else if(bCmdResetCarriageL)
						{
							gMachineFix.MoldL.Carriage.Zero = 0;
							gMachineFix.MoldL.Carriage.Max = 0;
							gRecipeOperate.OnceSave = 1;
							bCmdResetCarriageL = 0;
						}
						else if(bCmdResetBlowPin2R)
						{
							gMachineFix.MoldR.BlowPin2.Zero = 0;
							gMachineFix.MoldR.BlowPin2.Max = 0;
							gRecipeOperate.OnceSave = 1;
							bCmdResetBlowPin2R = 0;
						}
						else if(bCmdResetBlowPin2L)
						{
							gMachineFix.MoldL.BlowPin2.Zero = 0;
							gMachineFix.MoldL.BlowPin2.Max = 0;
							gRecipeOperate.OnceSave = 1;
							bCmdResetBlowPin2L = 0;
						}
						else if(bCmdResetExtrLift)
						{
							gMachineFix.ExtrLift.Zero = 0;
							gMachineFix.ExtrLift.Max = 0;
							gRecipeOperate.OnceSave = 1;
							bCmdResetExtrLift = 0;
						}
						uHideDiagResetCalib = 1;
						bCancelReset = 	0;
						bConfirmReset = 0;
					}
					else if (bCancelReset)
					{
						bCancelReset = 	0;
						bConfirmReset = 0;
						uHideDiagResetCalib = 1;
						bCmdResetClampR = 0;
						bCmdResetClampL = 0;
						bCmdResetBlowPinR = 0;
						bCmdResetBlowPinL = 0;
						bCmdResetBlowPin2R = 0;
						bCmdResetBlowPin2L = 0;
						bCmdResetCarriageR = 0;
						bCmdResetCarriageL = 0;
						bCmdResetExtrLift  =0;
					}
				}
				else
				{
					bCancelReset = 	0;
					bConfirmReset = 0;
					bCmdResetClampR = 0;
					bCmdResetClampL = 0;
					bCmdResetBlowPinR = 0;
					bCmdResetBlowPinL = 0;
					bCmdResetCarriageR = 0;
					bCmdResetCarriageL = 0;
					bCmdResetExtrLift  =0;
				}

				/*-------------------Calibration Confirm----------------------*/
				for(i=0;i<sizeof(CalibList)/2;i++)
				{
					CalibList[i] = 0;
				}

				CalibList[IndexCalib] = 1;

				gPanelObj.idxKeyPicture[S$KEYMATRIX_F13] = STATE_SUB_BUTTON;
					if(1 == gPanelObj.KeyMatric[S$KEYMATRIX_F13] && 1 == gTKcalib.Status)
					{
					cntF13 = cntF13 + 1;
				}
				else
				{
					cntF13 = 0;
				}

				if(cntF13 > 20)
				{
					if(1 == gMachineInfo.Calib && PIC_CALIB_CLAMP_ENCODER == gPanelObj.GetPicture )	/* 调校模式  */
					{
						switch(IndexCalib)
						{
							case 0:
								gMachineFix.MoldL.Clamp.Zero = LMold.Clamp.As;
								gRecipeOperate.OnceSave= 1;

								break;
							case 1:
								gMachineFix.MoldR.Clamp.Zero = RMold.Clamp.As;
								gRecipeOperate.OnceSave = 1;

								break;
							case 2:

								break;
							case 3:

								break;
							case 4:
								gMachineFix.MoldL.Clamp.Max = LMold.Clamp.As;
								gRecipeOperate.OnceSave = 1;

								break;

							case 5:
								gMachineFix.MoldR.Clamp.Max = RMold.Clamp.As;
								gRecipeOperate.OnceSave = 1;

								break;

							case 6:

								break;
							case 7:

								break;

						}/* switch(IndexCalib) */
					}/* if(1 == gMachineInfo.Calib)*/
					else if(1 == gMachineInfo.Calib && PIC_CALIB_CARRIAGE_ENCODER == gPanelObj.GetPicture)
					{
						switch(IndexCalib)
						{
							case 0:
								if(1 == LMold.TransDIn.CarriageFwLimit)
								{
									gMachineFix.MoldL.Carriage.Zero = LMold.Carriage.As;
									gRecipeOperate.OnceSave = 1;
								}
								else
								{
									gImply.LCarriageFw = 1;
								}
								break;
							case 1:
								if(1 == RMold.TransDIn.CarriageFwLimit)
								{
									gMachineFix.MoldR.Carriage.Zero = RMold.Carriage.As;
									gRecipeOperate.OnceSave = 1;
								}
								else
								{
									gImply.RCarriageFw = 1;
								}
								break;

							case 2:

								break;
							case 3:

								break;
							case 4:
								if(1 == LMold.TransDIn.CarriageBwLimit)
								{
									gMachineFix.MoldL.Carriage.Max = LMold.Carriage.As;
									gRecipeOperate.OnceSave = 1;
								}
								else
								{
									gImply.LCarriageBw = 1;
								}
								break;

							case 5:
								if(1 == RMold.TransDIn.CarriageBwLimit)
								{
									gMachineFix.MoldR.Carriage.Max = RMold.Carriage.As;
									gRecipeOperate.OnceSave = 1;
								}
								else
								{
									gImply.RCarriageBw = 1;
								}
								break;

							case 6:

								break;
							case 7:

								break;

						}/* switch(IndexCalib) */
					}
					else if(1 == gMachineInfo.Calib && PIC_CALIB_BLOWPIN_ENCODER == gPanelObj.GetPicture)
					{
						switch(IndexCalib)
						{
							case 0:
								if(1 == LMold.TransDIn.BlowPin2UpLimit)
								{
									gMachineFix.MoldL.BlowPin2.Zero = LMold.BlowPin2.As;
									gRecipeOperate.OnceSave = 1;
								}
								else
								{
									gImply.LPin2Up = 1;
								}
								break;
							case 1:
								if(1 == LMold.TransDIn.BlowPinUpLimit)
								{
									gMachineFix.MoldL.BlowPin.Zero = LMold.BlowPin.As;
									gRecipeOperate.OnceSave = 1;
								}
								else
								{
									gImply.LPinUp = 1;
								}
								break;

							case 2:
								if(1 == RMold.TransDIn.BlowPin2UpLimit)
								{
									gMachineFix.MoldR.BlowPin2.Zero = RMold.BlowPin2.As;
									gRecipeOperate.OnceSave = 1;
								}
								else
								{
									gImply.RPin2Up = 1;
								}
								break;
							case 3:
								if(1 == RMold.TransDIn.BlowPinUpLimit)
								{
									gMachineFix.MoldR.BlowPin.Zero = RMold.BlowPin.As;
									gRecipeOperate.OnceSave = 1;
								}
								else
								{
									gImply.RPinUp = 1;
								}
								break;
							case 4:
								gMachineFix.MoldL.BlowPin2.Max = LMold.BlowPin2.As;
								gRecipeOperate.OnceSave= 1;

								break;
							case 5:
								gMachineFix.MoldL.BlowPin.Max = LMold.BlowPin.As;
								gRecipeOperate.OnceSave = 1;

								break;

							case 6:
								gMachineFix.MoldR.BlowPin2.Max = RMold.BlowPin2.As;
								gRecipeOperate.OnceSave = 1;

								break;
							case 7:
								gMachineFix.MoldR.BlowPin.Max = RMold.BlowPin.As;
								gRecipeOperate.OnceSave = 1;

								break;

						}/* switch(IndexCalib) */
					}
					else if(1 == gMachineInfo.Calib && PIC_CALIB_OTHER_ENCODER == gPanelObj.GetPicture)
					{
						switch(IndexCalib)
						{
							case 0:

								break;
							case 1:
								if(1 == RMold.TransDIn.ExtruderLiftDnLimit)
								{
									gMachineFix.ExtrLift.Zero = RMold.ExtrLift.As;
									gRecipeOperate.OnceSave = 1;
								}
								else
								{
									gImply.ExtrLiftDn = 1;
								}

								break;

							case 2:

								break;
							case 3:

								break;
							case 4:

								break;
							case 5:
								//								if(1 == RMold.TransDIn.ExtruderLiftUpLimit)
								//								{
								gMachineFix.ExtrLift.Max = RMold.ExtrLift.As;
								gRecipeOperate.OnceSave = 1;
								//								}
								//								else
								//								{
								//									gImply.ExtrLiftUp = 1;
								//								}

								break;

							case 6:

								break;
							case 7:

								break;

						}/* switch(IndexCalib) */
					}
					else if(1 == gMachineInfo.Calib && PIC_CALIB_CLAMP_LVDT == gPanelObj.GetPicture)
					{
						switch(IndexCalib)
						{
							case 0:
								gMachineFix.MoldL.Clamp.Zero = LMold.Clamp.As;
								gRecipeOperate.OnceSave= 1;

								break;
							case 1:
								gMachineFix.MoldR.Clamp.Zero = RMold.Clamp.As;
								gRecipeOperate.OnceSave = 1;

								break;
							case 2:

								break;

							case 3:

								break;
							case 4:
								gMachineFix.MoldL.Clamp.Max = LMold.Clamp.As;
								gRecipeOperate.OnceSave = 1;

								break;
							case 5:
								gMachineFix.MoldR.Clamp.Max = RMold.Clamp.As;
								gRecipeOperate.OnceSave = 1;

								break;
							case 6:

								break;
							case 7:

								break;

						}/* switch(IndexCalib) */
					}
					else if(1 == gMachineInfo.Calib && PIC_CALIB_CARRIAGE_LVDT == gPanelObj.GetPicture)
					{
						switch(IndexCalib)
						{
							case 0:
								gMachineFix.MoldL.Carriage.Zero = LMold.Carriage.As;
								gRecipeOperate.OnceSave= 1;

								break;
							case 1:
								gMachineFix.MoldR.Carriage.Zero = RMold.Carriage.As;
								gRecipeOperate.OnceSave = 1;

								break;
							case 2:

								break;
							case 3:

								break;
							case 4:
								gMachineFix.MoldL.Carriage.Max = LMold.Carriage.As;
								gRecipeOperate.OnceSave = 1;

								break;
							case 5:
								gMachineFix.MoldR.Carriage.Max = RMold.Carriage.As;
								gRecipeOperate.OnceSave = 1;

								break;
							case 6:

								break;
							case 7:

								break;

						}/* switch(IndexCalib) */
					}
					else if(1 == gMachineInfo.Calib && PIC_CALIB_BLOWPIN_LVDT == gPanelObj.GetPicture)
					{
						switch(IndexCalib)
						{
							case 0:
								gMachineFix.MoldL.BlowPin.Zero = LMold.BlowPin.As;
								gRecipeOperate.OnceSave= 1;

								break;
							case 1:
								gMachineFix.MoldR.BlowPin.Zero = RMold.BlowPin.As;
								gRecipeOperate.OnceSave = 1;
								break;

							case 2:

								break;
							case 3:

								break;
							case 4:
								gMachineFix.MoldL.BlowPin.Max = LMold.BlowPin.As;
								gRecipeOperate.OnceSave = 1;

								break;

							case 5:
								gMachineFix.MoldR.BlowPin.Max = RMold.BlowPin.As;
								gRecipeOperate.OnceSave = 1;

								break;

							case 6:

								break;
							case 7:

								break;

						}/* switch(IndexCalib) */
					}
					else
					{
						gImply.CalMode = !gMachineInfo.Calib;
					}

				}/* if(1 == EDGEPOS(gPanelObj.KeyMatric[S$KEY_F13],KeyMatric[S$KEY_F13])) */

				// Robot Calib
				if(PIC_CALIB_ROBOT_ENCODER == gPanelObj.GetPicture)
				{
					if(1 == bRRobotHorZero)
					{
						cntRRobotHorZero++;
					}
					else
					{
						RMold.Robot.Transfer.Home = 0;
						cntRRobotHorZero =0;
					}

					if(1 == bRRobotVerZero)
					{
						RMold.Robot.UpDn.Home = 0;
						cntRRobotVerZero++;
					}
					else
					{
						cntRRobotVerZero =0;
					}

					if(1 == bLRobotHorZero)
					{
						cntLRobotHorZero++;
					}
					else
					{
						LMold.Robot.Transfer.Home = 0;
						cntLRobotHorZero =0;
					}

					if(1 == bLRobotVerZero)
					{
						cntLRobotVerZero++;
					}
					else
					{
						LMold.Robot.UpDn.Home =0;
						cntLRobotVerZero =0;
					}

					if(1 == gMachineInfo.Calib)	/* clibration mode  */
					{
						if(cntRRobotHorZero > 20)
						{
							if(1 == gMachineIn.RMold.RobotBwLimit)
							{
								gMachineFix.MoldR.RobotTransfer.sHome = RMold.Robot.Transfer.ecAs;
							}
							else
							{
								gImply.RRobotBw = 1;
							}
						}

						if(cntRRobotVerZero > 20)
						{
							if(1 == gMachineIn.RMold.RobotUpLimit)
							{
								gMachineFix.MoldR.RobotUpDn.sHome = RMold.Robot.UpDn.ecAs;
							}
							else
							{
								gImply.RRobotUp = 1;
							}
						}

						if(cntLRobotHorZero > 20)
						{
							if(1 == gMachineIn.LMold.RobotBwLimit)
							{
								gMachineFix.MoldL.RobotTransfer.sHome = LMold.Robot.Transfer.ecAs;
							}
							else
							{
								gImply.LRobotBw = 1;
							}
						}

						if(cntLRobotVerZero > 20)
						{
							if(1 == gMachineIn.LMold.RobotUpLimit)
							{
								gMachineFix.MoldL.RobotUpDn.sHome = LMold.Robot.UpDn.ecAs;
							}
							else
							{
								gImply.LRobotUp = 1;
							}
						}
					}
				}

				gPanelObj.idxKeyPicture[S$KEYMATRIX_F14] = STATE_INACTIVE;
					gPanelObj.idxKeyPicture[S$KEYMATRIX_F15] = STATE_INACTIVE;
					gPanelObj.idxKeyPicture[S$KEYMATRIX_F16] = STATE_SUB_PAGE;

					if(1 == EDGEPOS(gPanelObj.KeyMatric[S$KEYMATRIX_F16],KeyMatric[S$KEYMATRIX_F16]))
					{
					gPanelObj.SetPicture = PIC_PASSWORD_LOGIN;
				}
				break;

			case PIC_SCREEN_CALIBRATE:
				if(ChangePageDly > 0)
				{
					ChangePageDly--;
					break;
				}

				gPanelObj.idxKeyPicture[S$KEYMATRIX_F1] = STATE_SUB_PAGE;
					if(1 == EDGEPOS(gPanelObj.KeyMatric[S$KEYMATRIX_F1],KeyMatric[S$KEYMATRIX_F1]))
					{
					gPanelObj.SetPicture = PIC_OVERVIEW;
				}

				gPanelObj.idxKeyPicture[S$KEYMATRIX_F2] = STATE_SUB_PAGE;
					if(1 == EDGEPOS(gPanelObj.KeyMatric[S$KEYMATRIX_F2],KeyMatric[S$KEYMATRIX_F2]))
					{
					gPanelObj.SetPicture = gPanelObj.OldPicture;
				}

				gPanelObj.idxKeyPicture[S$KEYMATRIX_F3] = STATE_INACTIVE;
					gPanelObj.idxKeyPicture[S$KEYMATRIX_F4] = STATE_INACTIVE;
					gPanelObj.idxKeyPicture[S$KEYMATRIX_F5] = STATE_INACTIVE;
					gPanelObj.idxKeyPicture[S$KEYMATRIX_F6] = STATE_INACTIVE;
					gPanelObj.idxKeyPicture[S$KEYMATRIX_F7] = STATE_INACTIVE;
					gPanelObj.idxKeyPicture[S$KEYMATRIX_F8] = STATE_SUB_BUTTON;

					if(1 == EDGEPOS(gPanelObj.KeyMatric[S$KEYMATRIX_F8],KeyMatric[S$KEYMATRIX_F8]))
					{
					gPanelObj.vcHandle = VA_Setup(1, gPanelObj.VisualName);

					if (gPanelObj.vcHandle != 0)
					{
						if (!VA_Saccess(1, gPanelObj.vcHandle))
						{
							VA_StartTouchCal (1,gPanelObj.vcHandle);
							VA_Srelease(1, gPanelObj.vcHandle);
						}
					}
				}
				gPanelObj.idxKeyPicture[S$KEYMATRIX_F9] = STATE_INACTIVE;
					gPanelObj.idxKeyPicture[S$KEYMATRIX_F10] = STATE_INACTIVE;
					gPanelObj.idxKeyPicture[S$KEYMATRIX_F11] = STATE_INACTIVE;
					gPanelObj.idxKeyPicture[S$KEYMATRIX_F12] = STATE_INACTIVE;
					gPanelObj.idxKeyPicture[S$KEYMATRIX_F13] = STATE_INACTIVE;
					gPanelObj.idxKeyPicture[S$KEYMATRIX_F14] = STATE_INACTIVE;
					gPanelObj.idxKeyPicture[S$KEYMATRIX_F15] = STATE_INACTIVE;

					gPanelObj.idxKeyPicture[S$KEYMATRIX_F16] = STATE_SUB_PAGE;
					if(1 == EDGEPOS(gPanelObj.KeyMatric[S$KEYMATRIX_F16],KeyMatric[S$KEYMATRIX_F16]))
					{
					gPanelObj.SetPicture = PIC_PASSWORD_LOGIN;
				}
				if(ready == 0)
				{
					VC_HANDLE = VA_Setup(1 , gPanelObj.VisualName);

					if(VC_HANDLE != 0)ready = 1;
				}

				if(1 == ready)
				{
					if (!VA_Saccess(1,VC_HANDLE))
					{
						VA_GetTouchAction (1,VC_HANDLE,0,(UDINT)(&touch));
						VA_Ellipse (1,VC_HANDLE,touch.x,touch.y,2,2,0,0);
						VA_Srelease(1,VC_HANDLE);
					}
				}
				break;

			/*2018.8.3 Albert add new page for fast setting*/
			case PIC_FAST_SETTING:
				if(ChangePageDly > 0)
				{
					ChangePageDly--;
					break;
				}

				/*-----------F1---------*/
				gPanelObj.idxKeyPicture[S$KEYMATRIX_F1] = STATE_SUB_PAGE;
					if(1 == EDGEPOS(gPanelObj.KeyMatric[S$KEYMATRIX_F1],KeyMatric[S$KEYMATRIX_F1]))
					{
					gPanelObj.SetPicture = PIC_OVERVIEW;
				}
				/*-----------F2---------*/
				gPanelObj.idxKeyPicture[S$KEYMATRIX_F2] = STATE_SUB_PAGE;
					if(1 == EDGEPOS(gPanelObj.KeyMatric[S$KEYMATRIX_F2],KeyMatric[S$KEYMATRIX_F2]))
					{
					gPanelObj.SetPicture = gPanelObj.OldPicture;
				}
				/*-----------F3---------*/
				gPanelObj.idxKeyPicture[S$KEYMATRIX_F3] = STATE_SUB_PAGE;
					if(1 == bHideLeftStation)gPanelObj.idxKeyPicture[S$KEYMATRIX_F3] = STATE_INACTIVE;
					if(1 == EDGEPOS(gPanelObj.KeyMatric[S$KEYMATRIX_F3],KeyMatric[S$KEYMATRIX_F3]))
					{
					if(0 == bHideLeftStation)gPanelObj.SetPicture = PIC_CLAMP_L;
				}
				if(gPanelObj.GetPicture == PIC_CLAMP_L)gPanelObj.idxKeyPicture[S$KEYMATRIX_F3] = STATE_ACTIVE;

					/*-----------F4---------*/
					gPanelObj.idxKeyPicture[S$KEYMATRIX_F4] = STATE_SUB_PAGE;
					if(1 == EDGEPOS(gPanelObj.KeyMatric[S$KEYMATRIX_F4],KeyMatric[S$KEYMATRIX_F4]))
					{
					gPanelObj.SetPicture = PIC_CLAMP_R;
				}
				if(gPanelObj.GetPicture == PIC_CLAMP_R)gPanelObj.idxKeyPicture[S$KEYMATRIX_F4] = STATE_ACTIVE;

					/*-------------F5---------*/
					gPanelObj.idxKeyPicture[S$KEYMATRIX_F5] = STATE_SUB_PAGE;
					if(1 == bHideLeftStation)gPanelObj.idxKeyPicture[S$KEYMATRIX_F5] = STATE_INACTIVE;
					if(1 == EDGEPOS(gPanelObj.KeyMatric[S$KEYMATRIX_F5],KeyMatric[S$KEYMATRIX_F5]))
					{
					if(0 == bHideLeftStation)gPanelObj.SetPicture = PIC_TRANSPORT_L;
				}
				if(gPanelObj.GetPicture == PIC_TRANSPORT_L)gPanelObj.idxKeyPicture[S$KEYMATRIX_F5] = STATE_ACTIVE;

					/*------------F6-----------*/
					gPanelObj.idxKeyPicture[S$KEYMATRIX_F6] = STATE_SUB_PAGE;
					if(1 == EDGEPOS(gPanelObj.KeyMatric[S$KEYMATRIX_F6],KeyMatric[S$KEYMATRIX_F6]))
					{
					gPanelObj.SetPicture = PIC_TRANSPORT_R;
				}
				if(gPanelObj.GetPicture == PIC_TRANSPORT_R)gPanelObj.idxKeyPicture[S$KEYMATRIX_F6] = STATE_ACTIVE;

					/*------------F7-----------*/
					gPanelObj.idxKeyPicture[S$KEYMATRIX_F7] = STATE_SUB_PAGE;
					if(1 == bHideLeftStation)gPanelObj.idxKeyPicture[S$KEYMATRIX_F7] = STATE_INACTIVE;
					if(1 == EDGEPOS(gPanelObj.KeyMatric[S$KEYMATRIX_F7],KeyMatric[S$KEYMATRIX_F7]))
					{
					if(0 == bHideLeftStation)gPanelObj.SetPicture = PIC_BLOW_PIN_L;
				}
				if(gPanelObj.GetPicture == PIC_BLOW_PIN_L)gPanelObj.idxKeyPicture[S$KEYMATRIX_F7] = STATE_ACTIVE;

					/*-----------F8------------*/
					gPanelObj.idxKeyPicture[S$KEYMATRIX_F8] = STATE_SUB_PAGE;
					if(1 == EDGEPOS(gPanelObj.KeyMatric[S$KEYMATRIX_F8],KeyMatric[S$KEYMATRIX_F8]))
					{
					gPanelObj.SetPicture = PIC_BLOW_PIN_R;
				}
				if(gPanelObj.GetPicture == PIC_BLOW_PIN_R)gPanelObj.idxKeyPicture[S$KEYMATRIX_F8] = STATE_ACTIVE;

					/*----------F9-------------*/

					gPanelObj.idxKeyPicture[S$KEYMATRIX_F9] = STATE_SUB_PAGE;
					if(1 == EDGEPOS(gPanelObj.KeyMatric[S$KEYMATRIX_F9],KeyMatric[S$KEYMATRIX_F9]))
					{
					gPanelObj.SetPicture = PIC_DEFLASH;
				}
				if(gPanelObj.GetPicture == PIC_DEFLASH)gPanelObj.idxKeyPicture[S$KEYMATRIX_F9] = STATE_ACTIVE;

					/*----------F10-------------*/
					gPanelObj.idxKeyPicture[S$KEYMATRIX_F10] = STATE_INACTIVE;
					//						if(1 == EDGEPOS(gPanelObj.KeyMatric[S$KEYMATRIX_F10],KeyMatric[S$KEYMATRIX_F10]))
					//						{
					//						gPanelObj.SetPicture = PIC_BOTTOM_DEFLASH;
					//					}
					//					if(gPanelObj.GetPicture == PIC_BOTTOM_DEFLASH)gPanelObj.idxKeyPicture[S$KEYMATRIX_F10] = STATE_ACTIVE;

					gPanelObj.idxKeyPicture[S$KEYMATRIX_F11] = STATE_INACTIVE;
					//						if(1 == EDGEPOS(gPanelObj.KeyMatric[S$KEYMATRIX_F11],KeyMatric[S$KEYMATRIX_F11]))
					//						{
					//						gPanelObj.SetPicture = PIC_IO_DI_1;
					//					}

					gPanelObj.idxKeyPicture[S$KEYMATRIX_F12] = STATE_SUB_PAGE;
					if(1 == EDGEPOS(gPanelObj.KeyMatric[S$KEYMATRIX_F12],KeyMatric[S$KEYMATRIX_F12]))
					{
					gPanelObj.SetPicture = PIC_ALARM_CURRENT;
				}

				gPanelObj.idxKeyPicture[S$KEYMATRIX_F13] = STATE_SUB_PAGE;
					if(1 == EDGEPOS(gPanelObj.KeyMatric[S$KEYMATRIX_F13],KeyMatric[S$KEYMATRIX_F13]))
					{
					gPanelObj.SetPicture = PIC_AUTO_STEP;
				}

				gPanelObj.idxKeyPicture[S$KEYMATRIX_F14] = STATE_SUB_PAGE;
					if(1 == EDGEPOS(gPanelObj.KeyMatric[S$KEYMATRIX_F14],KeyMatric[S$KEYMATRIX_F14]))
					{
					gPanelObj.SetPicture = PIC_AUTO_START;
				}

				gPanelObj.idxKeyPicture[S$KEYMATRIX_F15] = STATE_SUB_PAGE;
					if(1 == EDGEPOS(gPanelObj.KeyMatric[S$KEYMATRIX_F15],KeyMatric[S$KEYMATRIX_F15]))
					{
					gPanelObj.SetPicture = PIC_SPC_CTRL;
				}

				gPanelObj.idxKeyPicture[S$KEYMATRIX_F16] = STATE_SUB_PAGE;
					if(1 == EDGEPOS(gPanelObj.KeyMatric[S$KEYMATRIX_F16],KeyMatric[S$KEYMATRIX_F16]))
					{
					gPanelObj.SetPicture = PIC_PASSWORD_LOGIN;
				}

				if(1 == EDGEPOS(gPanelObj.KeyMatric[S$KEYMATRIX_UP],KeyMatric[S$KEYMATRIX_UP]))
					{
					gPanelObj.SetLanguage = 1;
				}

				if(1 == EDGEPOS(gPanelObj.KeyMatric[S$KEYMATRIX_DOWN],KeyMatric[S$KEYMATRIX_DOWN]))
					{
					gPanelObj.SetLanguage = 0;
				}

				if(1 == EDGEPOS(gPanelObj.KeyMatric[S$KEYMATRIX_ESC],KeyMatric[S$KEYMATRIX_ESC]))
					{
					gPwd.PwdLevel = 0;
					gPanelObj.SetPicture = PIC_INIT;
				}

				//					/*Albert Machine Option*/
				//					for(i=0;i<OptionDis.Count;i++)
				//					{
				//						if(1 == HotSpot[i])
				//						{
				//							HotSpot[i]  = 0;
				//							if(0 == OptionDis.pHideSource[i])
				//							{
				//								OptionDis.Current = i;
				//								OptionDis.pSource[OptionDis.Current] = !OptionDis.pSource[OptionDis.Current];
				//								gRecipeOperate.DataSave = 1;
				//							}
				//						}
				//						OptionDis.Obj[i]= OptionDis.pSource[i];
				//					}

				break;

			default:
				break;

		}/* switch(gPanelObj.GetPicture) */
	}

	/* 离开DO DI AI AO MODULE 页面，强制复位  */
	//	if(((gPanelObj.GetPicture > PIC_IO_MODULE) || (gPanelObj.GetPicture < PIC_IO_DI_1))&&
	//		((OldGetPicture >= PIC_IO_DI_1       ) || (OldGetPicture < PIC_IO_MODULE      )))
	if(((gPanelObj.GetPicture > PIC_IO_MODULE) || (gPanelObj.GetPicture < PIC_IO_DO_2))&&
		((OldGetPicture >= PIC_IO_DO_2       ) || (OldGetPicture < PIC_IO_MODULE      ))&&
		gPanelObj.GetPicture !=PIC_SCREEN_SAVE &&
		gPanelObj.GetPicture !=PIC_PRESSURE_CALIBRATION )
	{
		memset(&gHardWare.DOForce[0],0,sizeof(gHardWare.DOForce));
		memset(&gHardWare.AOForce[0],0,sizeof(gHardWare.AOForce));
		gHardWare.AOForceNum = 19;
		btnTesetPQ = 0;
	}

	OldGetPicture = gPanelObj.GetPicture;

	KeyMatric[S$KEYMATRIX_F5] = gPanelObj.KeyMatric[S$KEYMATRIX_F5];
		KeyMatric[S$KEYMATRIX_F6] = gPanelObj.KeyMatric[S$KEYMATRIX_F6];
		KeyMatric[S$KEYMATRIX_F7] = gPanelObj.KeyMatric[S$KEYMATRIX_F7];
		KeyMatric[S$KEYMATRIX_F8] = gPanelObj.KeyMatric[S$KEYMATRIX_F8];

		/* 调校不合理，进入调教状态 */
		if((PIC_INIT_SET       == gPanelObj.GetPicture)||
		(PIC_GAP_CALIBRATE  == gPanelObj.GetPicture)||
		(PIC_ACCU_CALIBRATE == gPanelObj.GetPicture)
		)
	{
		gControlInfo.ControlStatus = S$STATUS_CALIBRATE;
		gAlarm.ParisonLinearCalErr = 0;
	}
	else
	{
		gControlInfo.ControlStatus = S$STATUS_AUTORUN;
		bHidePurge = 0;

		if(0 == gServoLinear.IsReady)
		{
			bHidePurge = 1;
			gControlInfo.ControlStatus = S$STATUS_NEED_CALIBRATE;

			if(1 == gThickProf.FunOption.Servo)
			{
				gAlarm.ParisonLinearCalErr = !gServoLinear.IsReady;
			}
			else
			{
				gAlarm.ParisonLinearCalErr = 0;
			}
		}
	}/* A|B|C */

	if((gServoLinear.Current < gServoLinear.ZeroPos - 1000  ) || (gServoLinear.Current > gServoLinear.MaxPos + 1000))
	{
		if(1 == gThickProf.FunOption.Servo && 1 == gServoLinear.IsReady)
		{
			gAlarm.ParisonValuebeyond = 1;
		}
		else
		{
			gAlarm.ParisonValuebeyond = 0;
		}
	}
	else
	{
		gAlarm.ParisonValuebeyond = 0;
	}

	gMachineInfo.ReceipeNum = gRecipeOperate.Index;

}/*  end of cycle  */

void InitOptionLists(void)
{

	/*=================================================Parison=================================================*/
	/*ActuatorType*/
	memset(uOptActorParison, 2, sizeof(uOptActorParison));
	uOptActorParison[ACTUATOR_UNDEFINED]  = 0;
	uOptActorParison[ACTUATOR_HYD]  	= 0;
	uOptActorParison[ACTUATOR_ELECTRIC]  = 0;

	/*=================================================Clamp=================================================*/
	/*ActuatorType*/
	memset(uOptActorClamp, 2, sizeof(uOptActorClamp));
	uOptActorClamp[ACTUATOR_UNDEFINED]  = 0;
	uOptActorClamp[ACTUATOR_HYD]  	= 0;
	uOptActorClamp[ACTUATOR_ELECTRIC]  = 0;

	/*PressueOutputType*/
	memset(uOptPresOutClamp, 2, sizeof(uOptPresOutClamp));
	uOptPresOutClamp[PRESSURE_OUTPUT_UNDEFINED]  	= 0;
	uOptPresOutClamp[PRESSURE_OUTPUT_SYSTEM_SINGLE]  = 0;

	/*FluxOutputType*/
	memset(uOptFluxOutClamp, 2, sizeof(uOptFluxOutClamp));
	uOptFluxOutClamp[FLUX_OUTPUT_UNDEFINED]  	= 0;
	uOptFluxOutClamp[FLUX_OUTPUT_SYSTEM_SINGLE]  = 0;
	uOptFluxOutClamp[FLUX_OUTPUT_PROP_VALVE_SINGLE]  = 0;
	uOptFluxOutClamp[FLUX_OUTPUT_NONE]  = 0;

	/*=================================================Carriage=================================================*/
	/*ActuatorType*/
	memset(uOptActorCarriage, 2, sizeof(uOptActorCarriage));
	uOptActorCarriage[ACTUATOR_UNDEFINED]  = 0;
	uOptActorCarriage[ACTUATOR_HYD]  	= 0;
	uOptActorCarriage[ACTUATOR_ELECTRIC]  = 0;

	/*PressueOutputType*/
	memset(uOptPresOutCarriage, 2, sizeof(uOptPresOutCarriage));
	uOptPresOutCarriage[PRESSURE_OUTPUT_UNDEFINED]  	= 0;
	uOptPresOutCarriage[PRESSURE_OUTPUT_SYSTEM_SINGLE]  = 0;

	/*FluxOutputType*/
	memset(uOptFluxOutCarriage, 2, sizeof(uOptFluxOutCarriage));
	uOptFluxOutCarriage[FLUX_OUTPUT_UNDEFINED]  	= 0;
	uOptFluxOutCarriage[FLUX_OUTPUT_SYSTEM_SINGLE]  = 0;
	uOptFluxOutCarriage[FLUX_OUTPUT_PROP_VALVE_SINGLE]  	= 0;
	uOptFluxOutCarriage[FLUX_OUTPUT_NONE]  = 0;

	/*=================================================BlowPin=================================================*/
	/*ActuatorType*/
	memset(uOptActorBlowPin, 2, sizeof(uOptActorBlowPin));
	uOptActorBlowPin[ACTUATOR_UNDEFINED]  = 0;
	uOptActorBlowPin[ACTUATOR_HYD]  	 = 0;
	uOptActorBlowPin[ACTUATOR_ELECTRIC]  = 0;

	/*PressueOutputType*/
	memset(uOptPresOutBlowPin, 2, sizeof(uOptPresOutBlowPin));
	uOptPresOutBlowPin[PRESSURE_OUTPUT_UNDEFINED]  	= 0;
	uOptPresOutBlowPin[PRESSURE_OUTPUT_SYSTEM_SINGLE]  = 0;

	/*FluxOutputType*/
	memset(uOptFluxOutBlowPin, 2, sizeof(uOptFluxOutBlowPin));
	uOptFluxOutBlowPin[FLUX_OUTPUT_UNDEFINED]  	= 0;
	uOptFluxOutBlowPin[FLUX_OUTPUT_SYSTEM_SINGLE]  = 0;
	uOptFluxOutBlowPin[FLUX_OUTPUT_PROP_VALVE_SINGLE]  	= 0;
	uOptFluxOutBlowPin[FLUX_OUTPUT_NONE]  = 0;

	/*=================================================Top Deflash=================================================*/
	/*ActuatorType*/
	memset(uOptActorTopDeflash, 2, sizeof(uOptActorTopDeflash));
	uOptActorTopDeflash[ACTUATOR_UNDEFINED]  = 0;
	uOptActorTopDeflash[ACTUATOR_HYD]  	= 0;
	uOptActorTopDeflash[ACTUATOR_PNEU]  = 0;

	/*PressueOutputType*/
	memset(uOptPresOutTopDeflash, 2, sizeof(uOptPresOutTopDeflash));
	uOptPresOutTopDeflash[PRESSURE_OUTPUT_UNDEFINED]  	= 0;
	uOptPresOutTopDeflash[PRESSURE_OUTPUT_SYSTEM_SINGLE]  = 0;
	uOptPresOutTopDeflash[PRESSURE_OUTPUT_ACC]  	= 0;

	/*FluxOutputType*/
	memset(uOptFluxOutTopDeflash, 2, sizeof(uOptFluxOutTopDeflash));
	uOptFluxOutTopDeflash[FLUX_OUTPUT_UNDEFINED]  	= 0;
	uOptFluxOutTopDeflash[FLUX_OUTPUT_SYSTEM_SINGLE]  = 0;
	uOptFluxOutTopDeflash[FLUX_OUTPUT_ACC]  	= 0;

	/*=================================================Bottom Deflash=================================================*/
	/*ActuatorType*/
	memset(uOptActorBottomDeflash, 2, sizeof(uOptActorBottomDeflash));
	uOptActorBottomDeflash[ACTUATOR_UNDEFINED]  = 0;
	uOptActorBottomDeflash[ACTUATOR_HYD]  	= 0;
	uOptActorBottomDeflash[ACTUATOR_PNEU]  = 0;

	/*PressueOutputType*/
	memset(uOptPresOutBottomDeflash, 2, sizeof(uOptPresOutBottomDeflash));
	uOptPresOutBottomDeflash[PRESSURE_OUTPUT_UNDEFINED]  	= 0;
	uOptPresOutBottomDeflash[PRESSURE_OUTPUT_SYSTEM_SINGLE]  = 0;
	uOptPresOutBottomDeflash[PRESSURE_OUTPUT_ACC]  	= 0;

	/*FluxOutputType*/
	memset(uOptFluxOutBottomDeflash, 2, sizeof(uOptFluxOutBottomDeflash));
	uOptFluxOutBottomDeflash[FLUX_OUTPUT_UNDEFINED]  	= 0;
	uOptFluxOutBottomDeflash[FLUX_OUTPUT_SYSTEM_SINGLE]  = 0;
	uOptFluxOutBottomDeflash[FLUX_OUTPUT_ACC]  	= 0;

	/*=================================================SubMold=================================================*/
	/*ActuatorType*/
	memset(uOptActorSubMold, 2, sizeof(uOptActorSubMold));
	uOptActorSubMold[ACTUATOR_UNDEFINED]  = 0;
	uOptActorSubMold[ACTUATOR_HYD]  	= 0;

	/*PressueOutputType*/
	memset(uOptPresOutSubMold, 2, sizeof(uOptPresOutSubMold));
	uOptPresOutSubMold[PRESSURE_OUTPUT_UNDEFINED]  	= 0;
	uOptPresOutSubMold[PRESSURE_OUTPUT_SYSTEM_SINGLE]  = 0;
	uOptPresOutSubMold[PRESSURE_OUTPUT_ACC]  	= 0;
	uOptPresOutSubMold[PRESSURE_OUTPUT_NONE]  	= 0;

	/*FluxOutputType*/
	memset(uOptFluxOutSubMold, 2, sizeof(uOptFluxOutSubMold));
	uOptFluxOutSubMold[FLUX_OUTPUT_UNDEFINED]  	= 0;
	uOptFluxOutSubMold[FLUX_OUTPUT_SYSTEM_SINGLE]  = 0;
	uOptFluxOutSubMold[FLUX_OUTPUT_ACC]  	= 0;
	uOptFluxOutSubMold[FLUX_OUTPUT_NONE]  	= 0;

	/*=================================================Plate=================================================*/
	/*ActuatorType*/
	memset(uOptActorPlate, 2, sizeof(uOptActorPlate));
	uOptActorPlate[ACTUATOR_UNDEFINED]  = 0;
	uOptActorPlate[ACTUATOR_HYD]  	= 0;

	/*PressueOutputType*/
	memset(uOptPresOutPlate, 2, sizeof(uOptPresOutPlate));
	uOptPresOutPlate[PRESSURE_OUTPUT_UNDEFINED]  	= 0;
	uOptPresOutPlate[PRESSURE_OUTPUT_SYSTEM_SINGLE]  = 0;
	uOptPresOutPlate[PRESSURE_OUTPUT_ACC]  	= 0;
	uOptPresOutPlate[PRESSURE_OUTPUT_NONE]  = 0;

	/*FluxOutputType*/
	memset(uOptFluxOutPlate, 2, sizeof(uOptFluxOutPlate));
	uOptFluxOutPlate[FLUX_OUTPUT_UNDEFINED]  	= 0;
	uOptFluxOutPlate[FLUX_OUTPUT_SYSTEM_SINGLE]  = 0;
	uOptFluxOutPlate[FLUX_OUTPUT_ACC]  	= 0;
	uOptFluxOutPlate[FLUX_OUTPUT_NONE]  = 0;

	/*=================================================ExtrLift=================================================*/
	/*ActuatorType*/
	memset(uOptActorExtrLift, 2, sizeof(uOptActorExtrLift));
	uOptActorExtrLift[ACTUATOR_UNDEFINED]  = 0;
	uOptActorExtrLift[ACTUATOR_HYD]  	   = 0;
	uOptActorExtrLift[ACTUATOR_ELECTRIC]   = 0;

	/*PressueOutputType*/
	memset(uOptPresOutExtrLift, 2, sizeof(uOptPresOutExtrLift));
	uOptPresOutExtrLift[PRESSURE_OUTPUT_UNDEFINED]  	= 0;
	uOptPresOutExtrLift[PRESSURE_OUTPUT_ACC_EXTRLIFT]  	= 0;
	uOptPresOutExtrLift[PRESSURE_OUTPUT_NONE]  	= 0;

	/*FluxOutputType*/
	memset(uOptFluxOutExtrLift, 2, sizeof(uOptFluxOutExtrLift));
	uOptFluxOutExtrLift[FLUX_OUTPUT_UNDEFINED]  	= 0;
	uOptFluxOutExtrLift[FLUX_OUTPUT_ACC_EXTRLIFT]  	= 0;
	uOptFluxOutExtrLift[FLUX_OUTPUT_NONE]  	= 0;

	/*=================================================Robot Transfer=================================================*/
	/*ActuatorType*/
	memset(uOptActorRobotTransfer, 2, sizeof(uOptActorRobotTransfer));
	uOptActorRobotTransfer[ACTUATOR_UNDEFINED]  = 0;
	uOptActorRobotTransfer[ACTUATOR_HYD]  	   = 0;
	uOptActorRobotTransfer[ACTUATOR_ELECTRIC]   = 0;
	uOptActorRobotTransfer[ACTUATOR_PNEU]    = 0;

	/*PressueOutputType*/
	memset(uOptPresOutRobotTransfer, 2, sizeof(uOptPresOutRobotTransfer));
	uOptPresOutRobotTransfer[PRESSURE_OUTPUT_UNDEFINED]  	= 0;
	uOptPresOutRobotTransfer[PRESSURE_OUTPUT_SYSTEM_SINGLE]  = 0;
	uOptPresOutRobotTransfer[PRESSURE_OUTPUT_NONE]  	= 0;

	/*FluxOutputType*/
	memset(uOptFluxOutRobotTranfer, 2, sizeof(uOptFluxOutRobotTranfer));
	uOptFluxOutRobotTranfer[FLUX_OUTPUT_UNDEFINED]  	= 0;
	uOptFluxOutRobotTranfer[FLUX_OUTPUT_SYSTEM_SINGLE]  = 0;
	uOptFluxOutRobotTranfer[FLUX_OUTPUT_NONE]  	= 0;

	/*=================================================Robot UpDn=================================================*/
	/*ActuatorType*/
	memset(uOptActorRobotUpDn, 2, sizeof(uOptActorRobotUpDn));
	uOptActorRobotUpDn[ACTUATOR_UNDEFINED]  = 0;
	uOptActorRobotUpDn[ACTUATOR_HYD]  	   = 0;
	uOptActorRobotUpDn[ACTUATOR_ELECTRIC]   = 0;
	uOptActorRobotUpDn[ACTUATOR_PNEU]    = 0;

	/*PressueOutputType*/
	memset(uOptPresOutRobotUpDn, 2, sizeof(uOptPresOutRobotUpDn));
	uOptPresOutRobotUpDn[PRESSURE_OUTPUT_UNDEFINED]  	= 0;
	uOptPresOutRobotUpDn[PRESSURE_OUTPUT_SYSTEM_SINGLE]  = 0;
	uOptPresOutRobotUpDn[PRESSURE_OUTPUT_NONE]  	= 0;

	/*FluxOutputType*/
	memset(uOptFluxOutRobotUpDn, 2, sizeof(uOptFluxOutRobotUpDn));
	uOptFluxOutRobotUpDn[FLUX_OUTPUT_UNDEFINED]  	= 0;
	uOptFluxOutRobotUpDn[FLUX_OUTPUT_SYSTEM_SINGLE]  = 0;
	uOptFluxOutRobotUpDn[FLUX_OUTPUT_NONE]  	= 0;

	/*=================================================Robot OpnCls=================================================*/
	/*ActuatorType*/
	memset(uOptActorRobotOpnCls, 2, sizeof(uOptActorRobotOpnCls));
	uOptActorRobotOpnCls[ACTUATOR_UNDEFINED]  = 0;
	uOptActorRobotOpnCls[ACTUATOR_HYD]  	   = 0;
	uOptActorRobotOpnCls[ACTUATOR_PNEU]   	= 0;

	/*PressueOutputType*/
	memset(uOptPresOutRobotOpnCls, 2, sizeof(uOptPresOutRobotOpnCls));
	uOptPresOutRobotOpnCls[PRESSURE_OUTPUT_UNDEFINED]  	= 0;
	uOptPresOutRobotOpnCls[PRESSURE_OUTPUT_SYSTEM_SINGLE]  = 0;
	uOptPresOutRobotOpnCls[PRESSURE_OUTPUT_NONE]  	= 0;

	/*FluxOutputType*/
	memset(uOptFluxOutRobotOpnCls, 2, sizeof(uOptFluxOutRobotOpnCls));
	uOptFluxOutRobotOpnCls[FLUX_OUTPUT_UNDEFINED]  	= 0;
	uOptFluxOutRobotOpnCls[FLUX_OUTPUT_SYSTEM_SINGLE]  = 0;
	uOptFluxOutRobotOpnCls[FLUX_OUTPUT_NONE]  	= 0;
}

void OptionListsUpdate(Mold_Fix_typ *pRMachineFix, Plate_Fix_typ *pPlateFix, ExtrLift_Fix_typ *pExtrLiftFix)
{
	UDINT old_Clamp_eActuatorType;
	/*=================================================Clamp=================================================*/
	/*ActuatorType*/
	if(ACTUATOR_HYD == pRMachineFix->Clamp.eActuatorType)  // Hydraulic
	{
		pRMachineFix->Clamp.eMechanismType = MECHANISM_LINEAR;
	}
	else if (ACTUATOR_ELECTRIC == pRMachineFix->Clamp.eActuatorType) // Electric
	{
		pRMachineFix->Clamp.eValveType 			= VALVE_UNDEFINED;
		pRMachineFix->Clamp.eSensorType 		= SENSOR_UNDEFINED;
		pRMachineFix->Clamp.ePressueOutputType 	= PRESSURE_OUTPUT_UNDEFINED;
		pRMachineFix->Clamp.eFluxOutputType 	= FLUX_OUTPUT_UNDEFINED;
	}
	else if (ACTUATOR_UNDEFINED == pRMachineFix->Clamp.eActuatorType) // Undefined
	{
		pRMachineFix->Clamp.eMechanismType = MECHANISM_LINEAR;
		pRMachineFix->Clamp.eValveType 			= VALVE_UNDEFINED;
		pRMachineFix->Clamp.eSensorType 		= SENSOR_UNDEFINED;
		pRMachineFix->Clamp.ePressueOutputType 	= PRESSURE_OUTPUT_UNDEFINED;
		pRMachineFix->Clamp.eFluxOutputType 	= FLUX_OUTPUT_UNDEFINED;
	}

	/*ValveType*/
	if(VALVE_PROP != pRMachineFix->Clamp.eValveType || ACTUATOR_HYD != pRMachineFix->Clamp.eActuatorType)  // Dir
	{
		gMachineFix.Option.bClampPropValveOutputInverse = 0;
	}

	/*=================================================Carriage=================================================*/
	/*ActuatorType*/
	if(ACTUATOR_HYD == pRMachineFix->Carriage.eActuatorType)  // Hydraulic
	{
		pRMachineFix->Carriage.eMechanismType = MECHANISM_LINEAR;
	}
	else if (ACTUATOR_ELECTRIC == pRMachineFix->Carriage.eActuatorType) // Electric
	{
		pRMachineFix->Carriage.eValveType 			= VALVE_UNDEFINED;
		pRMachineFix->Carriage.eSensorType 			= SENSOR_UNDEFINED;
		pRMachineFix->Carriage.ePressueOutputType 	= PRESSURE_OUTPUT_UNDEFINED;
		pRMachineFix->Carriage.eFluxOutputType 		= FLUX_OUTPUT_UNDEFINED;
	}
	else if (ACTUATOR_UNDEFINED == pRMachineFix->Carriage.eActuatorType) // Undefined
	{
		pRMachineFix->Carriage.eMechanismType = MECHANISM_LINEAR;
		pRMachineFix->Carriage.eValveType 			= VALVE_UNDEFINED;
		pRMachineFix->Carriage.eSensorType 			= SENSOR_UNDEFINED;
		pRMachineFix->Carriage.ePressueOutputType 	= PRESSURE_OUTPUT_UNDEFINED;
		pRMachineFix->Carriage.eFluxOutputType 	= FLUX_OUTPUT_UNDEFINED;
	}

	/*=================================================BlowPin=================================================*/
	/*ActuatorType*/
	if(ACTUATOR_HYD == pRMachineFix->BlowPin.eActuatorType)  // Hydraulic
	{
		pRMachineFix->BlowPin.eMechanismType = MECHANISM_LINEAR;
	}
	else if (ACTUATOR_ELECTRIC == pRMachineFix->BlowPin.eActuatorType) // Electric
	{
		pRMachineFix->BlowPin.eValveType 			= VALVE_UNDEFINED;
		pRMachineFix->BlowPin.eSensorType 			= SENSOR_UNDEFINED;
		pRMachineFix->BlowPin.ePressueOutputType 	= PRESSURE_OUTPUT_UNDEFINED;
		pRMachineFix->BlowPin.eFluxOutputType		= FLUX_OUTPUT_UNDEFINED;
	}
	else if (ACTUATOR_UNDEFINED == pRMachineFix->BlowPin.eActuatorType) // Undefined
	{
		pRMachineFix->BlowPin.eMechanismType = MECHANISM_LINEAR;
		pRMachineFix->BlowPin.eValveType 			= VALVE_UNDEFINED;
		pRMachineFix->BlowPin.eSensorType 			= SENSOR_UNDEFINED;
		pRMachineFix->BlowPin.ePressueOutputType 	= PRESSURE_OUTPUT_UNDEFINED;
		pRMachineFix->BlowPin.eFluxOutputType 	= FLUX_OUTPUT_UNDEFINED;
	}

	/*ValveType*/
	if(VALVE_PROP != pRMachineFix->BlowPin.eValveType || ACTUATOR_HYD != pRMachineFix->BlowPin.eActuatorType)  // Dir
	{
		gMachineFix.Option.bBlowpinPropValveOutputInverse = 0;
	}
	/*=================================================Top Deflash=================================================*/
	/*ActuatorType*/
	if(ACTUATOR_HYD == pRMachineFix->TopDeflash.eActuatorType)  // Hydraulic
	{
		//None
	}
	else if(ACTUATOR_PNEU == pRMachineFix->TopDeflash.eActuatorType) // Pneumatic
	{
		pRMachineFix->TopDeflash.ePressueOutputType = PRESSURE_OUTPUT_UNDEFINED;
		pRMachineFix->TopDeflash.eFluxOutputType 	= FLUX_OUTPUT_UNDEFINED;
	}
	else if (ACTUATOR_UNDEFINED == pRMachineFix->TopDeflash.eActuatorType) // Undefined
	{
		pRMachineFix->TopDeflash.ePressueOutputType = PRESSURE_OUTPUT_UNDEFINED;
		pRMachineFix->TopDeflash.eFluxOutputType 	= FLUX_OUTPUT_UNDEFINED;
	}

	/*=================================================Bottom Deflash=================================================*/
	/*ActuatorType*/
	if(ACTUATOR_HYD == pRMachineFix->BottomDeflash.eActuatorType)  // Hydraulic
	{
		//None
	}
	else if(ACTUATOR_PNEU == pRMachineFix->BottomDeflash.eActuatorType) // Pneumatic
	{
		pRMachineFix->BottomDeflash.ePressueOutputType 	= PRESSURE_OUTPUT_UNDEFINED;
		pRMachineFix->BottomDeflash.eFluxOutputType 	= FLUX_OUTPUT_UNDEFINED;
	}
	else if (ACTUATOR_UNDEFINED == pRMachineFix->BottomDeflash.eActuatorType) // Undefined
	{
		pRMachineFix->BottomDeflash.ePressueOutputType 	= PRESSURE_OUTPUT_UNDEFINED;
		pRMachineFix->BottomDeflash.eFluxOutputType 	= FLUX_OUTPUT_UNDEFINED;
	}

	/*=================================================SubMold=================================================*/
	/*ActuatorType*/
	if(ACTUATOR_HYD == pRMachineFix->SubMold.eActuatorType)  // Hydraulic
	{
		//None
	}
	else if (ACTUATOR_UNDEFINED == pRMachineFix->SubMold.eActuatorType) // Undefined
	{
		pRMachineFix->SubMold.ePressueOutputType 	= PRESSURE_OUTPUT_UNDEFINED;
		pRMachineFix->SubMold.eFluxOutputType 		= FLUX_OUTPUT_UNDEFINED;
	}

	/*=================================================Robot Transfer=================================================*/
	/*ActuatorType*/
	if(ACTUATOR_HYD == pRMachineFix->RobotTransfer.eActuatorType)  // Hydraulic
	{
		//None
	}
	else if(ACTUATOR_PNEU == pRMachineFix->RobotTransfer.eActuatorType) // Pneumatic
	{
		pRMachineFix->RobotTransfer.ePressueOutputType 	= PRESSURE_OUTPUT_UNDEFINED;
		pRMachineFix->RobotTransfer.eFluxOutputType 		= FLUX_OUTPUT_UNDEFINED;
	}
	else if (ACTUATOR_ELECTRIC == pRMachineFix->RobotTransfer.eActuatorType) // Electric
	{
		pRMachineFix->RobotTransfer.ePressueOutputType 	= PRESSURE_OUTPUT_UNDEFINED;
		pRMachineFix->RobotTransfer.eFluxOutputType 		= FLUX_OUTPUT_UNDEFINED;
	}
	else if (ACTUATOR_UNDEFINED == pRMachineFix->RobotTransfer.eActuatorType) // Undefined
	{
		pRMachineFix->RobotTransfer.ePressueOutputType 	= PRESSURE_OUTPUT_UNDEFINED;
		pRMachineFix->RobotTransfer.eFluxOutputType 		= FLUX_OUTPUT_UNDEFINED;
	}

	/*=================================================Robot UpDn=================================================*/
	/*ActuatorType*/
	if(ACTUATOR_HYD == pRMachineFix->RobotUpDn.eActuatorType)  // Hydraulic
	{
		//None
	}
	else if(ACTUATOR_PNEU == pRMachineFix->RobotUpDn.eActuatorType) // Pneumatic
	{
		pRMachineFix->RobotUpDn.ePressueOutputType 	= PRESSURE_OUTPUT_UNDEFINED;
		pRMachineFix->RobotUpDn.eFluxOutputType 		= FLUX_OUTPUT_UNDEFINED;
	}
	else if (ACTUATOR_UNDEFINED == pRMachineFix->RobotUpDn.eActuatorType) // Electric
	{
		pRMachineFix->RobotUpDn.ePressueOutputType 	= PRESSURE_OUTPUT_UNDEFINED;
		pRMachineFix->RobotUpDn.eFluxOutputType 		= FLUX_OUTPUT_UNDEFINED;
	}

	/*=================================================Robot OpnCls=================================================*/
	/*ActuatorType*/
	if(ACTUATOR_HYD == pRMachineFix->RobotOpnCls.eActuatorType)  // Hydraulic
	{
		//None
	}
	else if(ACTUATOR_PNEU == pRMachineFix->RobotOpnCls.eActuatorType) // Pneumatic
	{
		pRMachineFix->RobotOpnCls.ePressueOutputType 	= PRESSURE_OUTPUT_UNDEFINED;
		pRMachineFix->RobotOpnCls.eFluxOutputType 		= FLUX_OUTPUT_UNDEFINED;
	}
	else if (ACTUATOR_UNDEFINED == pRMachineFix->RobotOpnCls.eActuatorType) // Electric
	{
		pRMachineFix->RobotOpnCls.ePressueOutputType 	= PRESSURE_OUTPUT_UNDEFINED;
		pRMachineFix->RobotOpnCls.eFluxOutputType 		= FLUX_OUTPUT_UNDEFINED;
	}

	/*=================================================Plate=================================================*/
	/*ActuatorType*/
	if(ACTUATOR_HYD == pPlateFix->eActuatorType)  // Hydraulic
	{
		//None
	}
	else if (ACTUATOR_UNDEFINED == pPlateFix->eActuatorType) // Electric
	{
		pPlateFix->ePressueOutputType 	= PRESSURE_OUTPUT_UNDEFINED;
		pPlateFix->eFluxOutputType 		= FLUX_OUTPUT_UNDEFINED;
	}

	/*=================================================ExtrLift=================================================*/
	/*ActuatorType*/
	if(ACTUATOR_HYD == pExtrLiftFix->eActuatorType)  // Hydraulic
	{
		//None
	}
	else if(ACTUATOR_ELECTRIC == pExtrLiftFix->eActuatorType) // Electric
	{
		pExtrLiftFix->ePressueOutputType 	= PRESSURE_OUTPUT_UNDEFINED;
		pExtrLiftFix->eFluxOutputType 		= FLUX_OUTPUT_UNDEFINED;
	}
	else if (ACTUATOR_UNDEFINED == pExtrLiftFix->eActuatorType) // Electric
	{
		pExtrLiftFix->ePressueOutputType 	= PRESSURE_OUTPUT_UNDEFINED;
		pExtrLiftFix->eFluxOutputType 		= FLUX_OUTPUT_UNDEFINED;
	}

}
```

#### panel.typ - Local data types
```iecst
(********************************************************************
 * COPYRIGHT --
 ********************************************************************
 * Program: h_plan
 * File: h_plan.typ
 * Author: lij
 * Created: March 06, 2013
 ********************************************************************
 * Local data types of program h_plan
 ********************************************************************)

TYPE
	Object_Focus_typ : 	STRUCT
		Obj : ARRAY[0..MAX_OBJECT]OF UINT;
		Touch : ARRAY[0..MAX_OBJECT]OF USINT;
		pSource : REFERENCE TO USINT;
		pHideSource : REFERENCE TO USINT;
		Current : INT;
		Count : INT;
		Section : INT;
		Mode : INT;
	END_STRUCT;
END_TYPE
```

#### panel.var
```iecst
VAR
	cntTask : UDINT;
	bCmdTouch : BOOL;
	bHideFunctionKey : USINT;
	bHideVisu : USINT;
	bHideNoUse : USINT;
	bHidePurge : UINT;
	bHideFrame : UINT;
	bHidePropValvePage : UINT;
	bHideCarriagePropValve : UINT;
	bHideClampPropValve : UINT;
	bHideBlowPinPropValve : UINT;
	bHideParisonAutoCalib : UINT;
	bHideRSupportAirTimeVersion : USINT;
	bHideLSupportAirTimeVersion : USINT;
	bHideRSupportAir2TimeVersion : USINT;
	bHideLSupportAir2TimeVersion : USINT;
	bHideWordSupportAirTimeVersion : USINT;
	bHideWordSupportAir2TimeVersion : USINT;
	bHideRSupportSuckAirTimeVersion : USINT;
	bHideLSupportSuckAirTimeVersion : USINT;
	bHideWordSupportSuckAirTimeVer : USINT;
	bHideExtruderVFCtrl : USINT;
	bHideExtruderVFCtrlPara : USINT;
	bHideExtrA_VFCtrlPara : USINT;
	bHideExtrB_VFCtrlPara : USINT;
	bHideExtrC_VFCtrlPara : USINT;
	bHideExtrD_VFCtrlPara : USINT;
	bHideExtrV_VFCtrlPara : USINT;
END_VAR
(*HideClamp*)
VAR
	bHideClampActuatorElectic : USINT;
	bHideClampActuatorHyd : USINT;
	bHideRClampActuatorHyd : USINT;
	bHideLClampActuatorHyd : USINT;
	bHideClampActuatorHyd_LVDT : USINT;
	bHideClampActuatorHyd_Switch : USINT;
	bHideClampFluxOutput : USINT;
END_VAR
(*HideBlowPin*)
VAR
	bHideBlowPinActuatorElectic : USINT;
	bHideBlowPinActuatorHyd : USINT;
	bHideBlowPinActuatorHyd_LVDT : USINT;
	bHideBlowPinActuatorHyd_Switch : USINT;
	bHideLBlowPinActuatorHyd_Switch : USINT;
	bHideBlowPinFluxOutput : USINT;
END_VAR
(*HideCarriage*)
VAR
	bHideCarriageActuatorElectic : USINT;
	bHideCarriageActuatorHyd : USINT;
	bHideRCarriageActuatorHyd : USINT;
	bHideLCarriageActuatorHyd : USINT;
	bHideCarriageActuatorHyd_LVDT : USINT;
	bHideCarriageActuatorHyd_Switch : USINT;
	bHideLCarriageActuatorHyd_Switch : USINT;
	bHideCarriageFluxOutput : USINT;
END_VAR
(*HideTopDeflash*)
VAR
	bHideTopDeflashActuatorHyd : USINT;
	bHideRTopDeflashPresOutput : USINT;
	bHideRTopDeflashFluxOutput : USINT;
	bHideLTopDeflashPresOutput : USINT;
	bHideLTopDeflashFluxOutput : USINT;
END_VAR
(*HideBottomDeflash*)
VAR
	bHideBottomDeflashActuatorHyd : USINT;
	bHideRBottomDeflashPresOutput : USINT;
	bHideRBottomDeflashFluxOutput : USINT;
	bHideLBottomDeflashPresOutput : USINT;
	bHideLBottomDeflashFluxOutput : USINT;
END_VAR
(*HideExtrLift*)
VAR
	bHideExtrLiftActuatorHyd : USINT;
	bHideRExtrLiftActuatorHyd : USINT;
	bHideLExtrLiftActuatorHyd : USINT;
	bHideExtrLiftActuatorElectric : USINT;
	bHideExtrLiftPresOutput : USINT;
	bHideExtrLiftFluxOutput : USINT;
END_VAR
(*HideSubmold*)
VAR
	bHideSubmoldActuatorHyd : USINT;
	bHideRSubMoldPresOutput : USINT;
	bHideRSubMoldFluxOutput : USINT;
	bHideLSubMoldPresOutput : USINT;
	bHideLSubMoldFluxOutput : USINT;
END_VAR
(*Hide Plate*)
VAR
	bHidePlateActuatorHyd : USINT;
	bHidePlateUpDnPresOutput : USINT;
	bHidePlateUpDnFluxOutput : USINT;
	bHidePlateFwBwPresOutput : USINT;
	bHidePlateFwBwFluxOutput : USINT;
END_VAR
(*HideRobotTransfer*)
VAR
	bHideRobotTransferActuatorHyd : USINT;
	bHideRobotTransferActuatorElec : USINT;
	bHideRobotTransferActuatorPneu : USINT;
	bHideRobotUpDnActuatorHyd : USINT;
	bHideRobotUpDnActuatorElectric : USINT;
	bHideRobotUpDnActuatorPneu : USINT;
	bHideRobotOpnClsActuatorHyd : USINT;
	bHideRobotOpnClsActuatorPneu : USINT;
	bHideAutoLubr : USINT;
	MarkerDis : Object_Focus_typ;
	OptionDis : Object_Focus_typ;
	OptionWordHide : Option_typ;
	OptionHide : Machine_Option_typ;
	MacOptionOld : Machine_Option_typ;
	KeyMatric : ARRAY[0..MAX_KEY_COUNT] OF USINT;
	OldSet : Share_Set_typ;
	OldFunSet : Thick_Function_typ;
	FLed : ARRAY[0..9] OF USINT;
	OldIsOpt : USINT;
	i : INT;
	Led : USINT;
	OldStation : USINT;
	IndexDo : INT;
	DoColor : ARRAY[0..199] OF UINT;
	InputColor : UINT;
	HotSpot : ARRAY[0..32] OF UINT;
	ready : UINT;
	touch : TouchAction;
	VC_HANDLE : UDINT;
	AoColor : ARRAY[0..19] OF UINT;
	IndexAo : INT;
	Zero : ARRAY[0..3] OF INT;
	Max : ARRAY[0..3] OF INT;
	IndexCalib : INT;
	CalibList : ARRAY[0..15] OF INT;
	ChangePageDly : UDINT;
	bTimeRtoL : USINT;
	OldGetPicture : UINT;
	bHideForceDO : UINT;
	bAutoHide : UINT;
	bTimeLtoR : USINT;
	bZoneHide : ARRAY[0..MAX_IDX_ZONE] OF UINT;
	bOEMZoneOptionHide : ARRAY[0..MAX_IDX_ZONE] OF UINT;
	bHideLeftStation : UINT;
	bHideParison : UINT;
	bHideParisonActuatorElectic : USINT;
	bHideParisonActuatorHyd : USINT;
	bHideBlowUpDuringClampCls : USINT;
	bHideWordTopDeflashAirOpt : USINT;
	bHideRTopDeflashAirOpt : USINT;
	bHideLTopDeflashAirOpt : USINT;
	bHideWordBottomDeflashAirOpt : USINT;
	bHideRBottomDeflashAirOpt : USINT;
	bHideLBottomDeflashAirOpt : USINT;
	bHideWordCoolBlow : USINT;
	bHideRCoolBlow : USINT;
	bHideLCoolBlow : USINT;
	bHideWordCoolBlow2 : USINT;
	bHideRCoolBlow2 : USINT;
	bHideLCoolBlow2 : USINT;
	bHideWordCoolBlow3 : USINT;
	bHideRCoolBlow3 : USINT;
	bHideLCoolBlow3 : USINT;
	bThickCalibHide : UINT;
	bLevel3CalibHide : USINT;
	bLevel4CalibHide : USINT;
	bHideACCPump : USINT;
	bHideACCPump_Extrlift : USINT;
	bHideHighPrsMotor : USINT;
	bHideCutterHeating : USINT;
	bHideDieLip : ARRAY[0..7] OF USINT;
	cntF7 : UDINT;
	cntF13 : UDINT;
	cntF8 : UDINT;
	bHideForceAO : UINT;
	idxZone : USINT;
	QuickSetValueFoucs : UINT;
	HeatingPlanFoucs : ARRAY[0..13] OF UINT;
	TempEnableFoucs : ARRAY[0..MAX_IDX_ZONE] OF UINT;
	bLRobotVerZero : BOOL;
	bLRobotHorZero : BOOL;
	bRRobotVerZero : BOOL;
	bRRobotHorZero : BOOL;
	cntLRobotHorZero : UINT;
	cntLRobotVerZero : UINT;
	cntRRobotHorZero : UINT;
	cntRRobotVerZero : UINT;
	BtnHeadA : USINT;
	BtnHeadAOld : USINT;
	BtnHeadAB : USINT;
	BtnHeadABOld : USINT;
	BtnHeadABC : USINT;
	BtnHeadABCOld : USINT;
END_VAR
(*Reset Calibrate Function*)
VAR
	uHideDiagResetCalib : USINT;
	bCmdResetExtrLift : BOOL;
	bCmdResetClampR : BOOL;
	bCmdResetClampL : BOOL;
	bCmdResetBlowPinR : BOOL;
	bCmdResetBlowPinL : BOOL;
	bCmdResetBlowPin2R : BOOL;
	bCmdResetBlowPin2L : BOOL;
	bCmdResetCarriageR : BOOL;
	bCmdResetCarriageL : BOOL;
	bConfirmReset : BOOL;
	bCancelReset : BOOL;
	OldLBottomSubMold : USINT;
	OldLSubMold : USINT;
	OldRBottomSubMold : USINT;
	OldRSubMold : USINT;
	bLBottomSubMold : USINT;
	bLSubMold : USINT;
	bRBottomSubMold : USINT;
	bRSubMold : USINT;
	bLCoolPin2 : USINT;
	bRCoolPin2 : USINT;
	bLCoolPin3 : USINT;
	bRCoolPin3 : USINT;
	bHideSealGap : USINT;
	bExtrA_Hide : USINT;
	bExtrB_Hide : USINT;
	bExtrC_Hide : USINT;
	bExtrD_Hide : USINT;
	bExtrV_Hide : USINT;
END_VAR
(*Parison Option*)
VAR
	uOptActorParison : ARRAY[0..3] OF USINT := [4(0)];
END_VAR
(*Clamp Option*)
VAR
	uOptActorClamp : ARRAY[0..3] OF USINT := [4(0)];
	uOptPresOutClamp : ARRAY[0..4] OF USINT := [5(0)];
	uOptFluxOutClamp : ARRAY[0..5] OF USINT := [6(0)];
END_VAR
(*Carriage Option*)
VAR
	uOptActorCarriage : ARRAY[0..3] OF USINT := [4(0)];
	uOptPresOutCarriage : ARRAY[0..4] OF USINT := [5(0)];
	uOptFluxOutCarriage : ARRAY[0..5] OF USINT := [6(0)];
END_VAR
(*BlowPin Option*)
VAR
	uOptActorBlowPin : ARRAY[0..3] OF USINT := [4(0)];
	uOptPresOutBlowPin : ARRAY[0..4] OF USINT := [5(0)];
	uOptFluxOutBlowPin : ARRAY[0..5] OF USINT := [6(0)];
END_VAR
(*SubMold Option*)
VAR
	uOptActorSubMold : ARRAY[0..3] OF USINT := [4(0)];
	uOptPresOutSubMold : ARRAY[0..4] OF USINT := [5(0)];
	uOptFluxOutSubMold : ARRAY[0..5] OF USINT := [6(0)];
END_VAR
(*ExtrLift Option*)
VAR
	uOptActorExtrLift : ARRAY[0..3] OF USINT := [4(0)];
	uOptPresOutExtrLift : ARRAY[0..4] OF USINT := [5(0)];
	uOptFluxOutExtrLift : ARRAY[0..5] OF USINT := [6(0)];
END_VAR
(*Plate Option*)
VAR
	uOptActorPlate : ARRAY[0..3] OF USINT := [4(0)];
	uOptPresOutPlate : ARRAY[0..4] OF USINT := [5(0)];
	uOptFluxOutPlate : ARRAY[0..5] OF USINT := [6(0)];
END_VAR
(*Top Deflash Option*)
VAR
	uOptActorTopDeflash : ARRAY[0..3] OF USINT := [4(0)];
	uOptPresOutTopDeflash : ARRAY[0..4] OF USINT := [5(0)];
	uOptFluxOutTopDeflash : ARRAY[0..5] OF USINT := [6(0)];
END_VAR
(*Bottom Deflash Option*)
VAR
	uOptActorBottomDeflash : ARRAY[0..3] OF USINT := [4(0)];
	uOptPresOutBottomDeflash : ARRAY[0..4] OF USINT := [5(0)];
	uOptFluxOutBottomDeflash : ARRAY[0..5] OF USINT := [6(0)];
END_VAR
(*Robot Transfer Option*)
VAR
	uOptActorRobotTransfer : ARRAY[0..3] OF USINT := [4(0)];
	uOptPresOutRobotTransfer : ARRAY[0..4] OF USINT := [5(0)];
	uOptFluxOutRobotTranfer : ARRAY[0..5] OF USINT := [6(0)];
END_VAR
(*Robot UpDn Option*)
VAR
	uOptActorRobotUpDn : ARRAY[0..3] OF USINT := [4(0)];
	uOptPresOutRobotUpDn : ARRAY[0..4] OF USINT := [5(0)];
	uOptFluxOutRobotUpDn : ARRAY[0..5] OF USINT := [6(0)];
END_VAR
(*Robot OpnCls Option*)
VAR
	uOptActorRobotOpnCls : ARRAY[0..3] OF USINT := [4(0)];
	uOptPresOutRobotOpnCls : ARRAY[0..4] OF USINT := [5(0)];
	uOptFluxOutRobotOpnCls : ARRAY[0..5] OF USINT := [6(0)];
	keyF5N : USINT;
	keyF6N : USINT;
END_VAR
(*Index*)
VAR
	Index : USINT;
END_VAR
```

- thick.h (reference to Logical/GlobalIncludes/thick.h)

- pic_id.h (reference to Logical/GlobalIncludes/pic_id.h)

- defines.h (reference to Logical/GlobalIncludes/defines.h)

- keyap880.h (reference to Logical/GlobalIncludes/keyap880.h)

- keyap2100.h (reference to Logical/GlobalIncludes/keyap2100.h)

### Program Logical/screen/hmi_cpy (ANSIC, version 1.00.0) - auto copy screen to bmp file

#### hmi_cpy.c - Implementation code
```c
/********************************************************************
 * COPYRIGHT -- B&R Automation China
 ********************************************************************
 * Program: hmi_cpy
 * File: hmi_cpy.c
 * Author: lijianjun
 * Created: May 27, 2015
 ********************************************************************
 * Implementation of program hmi_cpy
 ********************************************************************/

#include <bur/plctypes.h>

#ifdef _DEFAULT_INCLUDES
	#include <AsDefault.h>
#endif

#include "pic_id.h"

void _INIT hmi_cpyINIT(void)
{
	/* TODO: Add code here */
   StepCopyScreen = 0;

   /* ----- get task cycle time ----- */
   RTInfo_Task.enable = 1;
   RTInfo(&RTInfo_Task);

   tTask = RTInfo_Task.cycle_time/1000.0/1000.0;		/*  from us ---> s  */
}

void _CYCLIC hmi_cpyCYCLIC(void)
{

   /* there is insert USB disk */
   if(1 == gRecipeOperate.usbDiskOk)
   {
      if(0 == StepCopyScreen)
      {
         if(1 == gScreenShot.CmdScreenShotAll)
         {
            gScreenShot.CmdScreenShotAll = 0;
            StepCopyScreen = 100;
         }
      }
      else
      {
         gScreenShot.CmdScreenShotAll = 0;
      }
   }
   else
   {
      if(1 == gScreenShot.CmdScreenShotAll)
      {
         gImply.NoUSB = 1;
         gScreenShot.CmdScreenShotAll = 0;
      }
      StepCopyScreen = 0;
      idxPicture = 0;
   }

   /* ------ step machine control ------ */
   switch(StepCopyScreen)
   {
      case 0:
         gScreenShot.ScreenShotRun = 0;
         tTimeOut = 0.0;
         break;

      /* change to first picture  */
      case 100:
         gScreenShot.ScreenShotRun = 1;
         idxPicture = PIC_OVERVIEW;      /* first picture --- PIC_OVERVIEW   */
         tTimeOut = 0.0;
         if(gPanelObj.GetPicture != PIC_OVERVIEW)
         {
            gPanelObj.SetPicture = PIC_OVERVIEW;
         }
         StepCopyScreen = 200;
         break;

      /*  change picture success or false  */
      case 200:
         tTimeOut = tTimeOut + tTask;
         if(idxPicture == gPanelObj.GetPicture)
         {
            StepCopyScreen = 300;
         }

         if(tTimeOut > 3.0)      /* change timeout reach */
         {
            tTimeOut = 0.0;
            StepCopyScreen = 600;
         }
         break;

      /* change picture ok then send screen shot command  */
      case 300:
         tTimeOut = 0.0;
         gScreenShot.CmdScreenShot = 1;
         StepCopyScreen = 400;
         break;

      case 400:
         tTimeOut = tTimeOut + tTask;

         if(tTimeOut > 0.5)
         {
            if(0 == gScreenShot.CmdScreenShot)
            {
               if(1 == gScreenShot.Status)
               {
                  tTimeOut = 0.0;
                  StepCopyScreen = 600;
               }
               else if(3 == gScreenShot.Status)
               {
                  tTimeOut = 0.0;
                  StepCopyScreen = 500;
               }
            }
         }

         if(tTimeOut > 20.0)      /* screen shot timeout reach */
         {
            tTimeOut = 0.0;
            gImply.ScreenShotFalse = 1;  /* screen shot error */
            StepCopyScreen = 3000;
         }
         break;

      /* screen shot flase then send command again  */
      case 500:
         if(1 == gScreenShot.Status)
         {
            tTimeOut = 0.0;
            StepCopyScreen = 300;
         }
         break;

      /* screen shot ok then change to next picture */
      case 600:
         tTimeOut = 0.0;
       // if(idxPicture < PIC_GAP_CALIBRATE_HELP + 1)
		if(idxPicture < PIC_FAST_SETTING + 1)  //ipis1227

         {
            idxPicture = idxPicture + 1;
            gPanelObj.SetPicture = idxPicture;
            StepCopyScreen = 200;
         }
         else
         {
            gPanelObj.SetPicture = 1;
            StepCopyScreen = 3000;
         }
         break;

      case 3000:
         gScreenShot.ScreenShotRun = 0;
         StepCopyScreen = 0;
         break;
   }/* switch(StepCopyScreen) */

}

void _EXIT hmi_cpyEXIT(void)
{
	/* TODO: Add code here */
}
```

#### hmi_cpy.var - Local variables
```iecst
(********************************************************************
 * COPYRIGHT --
 ********************************************************************
 * Program: hmi_cpy
 * File: hmi_cpy.var
 * Author: lij
 * Created: May 27, 2015
 ********************************************************************
 * Local variables of program hmi_cpy
 ********************************************************************)
VAR
	tTask : REAL := 0.0;
	RTInfo_Task : RTInfo := (0);
	tTimeOut : REAL;
	idxPicture : UINT;
	StepCopyScreen : UINT;
END_VAR
```

- pic_id.h (reference to Logical/GlobalIncludes/pic_id.h)

### Program Logical/screen/Trace (IEC)

#### Cyclic.st - Cyclic code
```iecst
(*********************************************************************************
 * Copyright: Bernecker+Rainer
 * Author:    ho2c
 * Created:   September 4, 2019/9:59 AM
 *********************************************************************************)

PROGRAM _CYCLIC
	(* Insert code here *)
	//----------------------
	//修改此處
	//----------------------
	//Data -> Struct

//	rData[0]	:= TraceData.rPosition;
//	rData[1]	:= TraceData.rSpeed;
//	rData[2]	:= TraceData.rTorque;
//	rData[3]	:= TraceData.rCurrent;

	IF 0=uMotorIndex THEN //RClamp
		rData[0]	:= gMotorTrace.RMold.Clamp.Position;
		rData[1]	:= gMotorTrace.RMold.Clamp.RPM;
		rData[2]	:= gMotorTrace.RMold.Clamp.Current;
		rData[3]	:= gMotorTrace.RMold.Clamp.Torque;
		Max_Torque	:= gMotorTrace.RMold.Clamp.Max_Torque_Set;
	END_IF;

	IF 1=uMotorIndex THEN //LClamp
		rData[0]	:= gMotorTrace.LMold.Clamp.Position;
		rData[1]	:= gMotorTrace.LMold.Clamp.RPM;
		rData[2]	:= gMotorTrace.LMold.Clamp.Current;
		rData[3]	:= gMotorTrace.LMold.Clamp.Torque;
		Max_Torque	:= gMotorTrace.LMold.Clamp.Max_Torque_Set;
	END_IF;

	IF 2=uMotorIndex THEN // RCarriage
		rData[0]	:= gMotorTrace.RMold.Carriage.Position;
		rData[1]	:= gMotorTrace.RMold.Carriage.RPM;
		rData[2]	:= gMotorTrace.RMold.Carriage.Current;
		rData[3]	:= gMotorTrace.RMold.Carriage.Torque;
		Max_Torque	:= gMotorTrace.RMold.Carriage.Max_Torque_Set;
	END_IF;

	IF 3=uMotorIndex THEN // LCarriage
		rData[0]	:= gMotorTrace.LMold.Carriage.Position;
		rData[1]	:= gMotorTrace.LMold.Carriage.RPM;
		rData[2]	:= gMotorTrace.LMold.Carriage.Current;
		rData[3]	:= gMotorTrace.LMold.Carriage.Torque;
		Max_Torque	:= gMotorTrace.LMold.Carriage.Max_Torque_Set;
	END_IF;

	IF 4=uMotorIndex THEN // RBlowpin1
		rData[0]	:= gMotorTrace.RMold.BlowPin.Position;
		rData[1]	:= gMotorTrace.RMold.BlowPin.RPM;
		rData[2]	:= gMotorTrace.RMold.BlowPin.Current;
		rData[3]	:= gMotorTrace.RMold.BlowPin.Torque;
		Max_Torque	:= gMotorTrace.RMold.BlowPin.Max_Torque_Set;
	END_IF;

	IF 5=uMotorIndex THEN // LBlowpin1
		rData[0]	:= gMotorTrace.LMold.BlowPin.Position;
		rData[1]	:= gMotorTrace.LMold.BlowPin.RPM;
		rData[2]	:= gMotorTrace.LMold.BlowPin.Current;
		rData[3]	:= gMotorTrace.LMold.BlowPin.Torque;
		Max_Torque	:= gMotorTrace.LMold.BlowPin.Max_Torque_Set;
	END_IF;

	IF 6=uMotorIndex THEN // RRobotTransfer
		rData[0]	:= gMotorTrace.RMold.RobotTransfer.Position;
		rData[1]	:= gMotorTrace.RMold.RobotTransfer.RPM;
		rData[2]	:= gMotorTrace.RMold.RobotTransfer.Current;
		rData[3]	:= gMotorTrace.RMold.RobotTransfer.Torque;
		Max_Torque	:= gMotorTrace.RMold.RobotTransfer.Max_Torque_Set;
	END_IF;

	IF 7=uMotorIndex THEN // LRobotTransfer
		rData[0]	:= gMotorTrace.LMold.RobotTransfer.Position;
		rData[1]	:= gMotorTrace.LMold.RobotTransfer.RPM;
		rData[2]	:= gMotorTrace.LMold.RobotTransfer.Current;
		rData[3]	:= gMotorTrace.LMold.RobotTransfer.Torque;
		Max_Torque	:= gMotorTrace.LMold.RobotTransfer.Max_Torque_Set;
	END_IF;

	IF 10=uMotorIndex THEN // Extrlift
		rData[0]	:= gMotorTrace.Extrlift.Position;
		rData[1]	:= gMotorTrace.Extrlift.RPM;
		rData[2]	:= gMotorTrace.Extrlift.Current;
		rData[3]	:= gMotorTrace.Extrlift.Torque;
		Max_Torque	:= gMotorTrace.Extrlift.Max_Torque_Set;
	END_IF;

	IF 11=uMotorIndex THEN // Parison
		rData[0]	:= gMotorTrace.Parison.Position;
		rData[1]	:= gMotorTrace.Parison.RPM;
		rData[2]	:= gMotorTrace.Parison.Current;
		rData[3]	:= gMotorTrace.Parison.Torque;
		Max_Torque	:= gMotorTrace.Parison.Max_Torque_Set;
	END_IF;

//	IF 14=uMotorIndex THEN // RBlowpin2
//		rData[0]	:= gMotorTrace.RMold.BlowPin2.Position;
//		rData[1]	:= gMotorTrace.RMold.BlowPin2.RPM;
//		rData[2]	:= gMotorTrace.RMold.BlowPin2.Current;
//		rData[3]	:= gMotorTrace.RMold.BlowPin2.Torque;
//	END_IF;
//
//	IF 15=uMotorIndex THEN //LBlowpin2
//		rData[0]	:= gMotorTrace.LMold.BlowPin2.Position;
//		rData[1]	:= gMotorTrace.LMold.BlowPin2.RPM;
//		rData[2]	:= gMotorTrace.LMold.BlowPin2.Current;
//		rData[3]	:= gMotorTrace.LMold.BlowPin2.Torque;
//	END_IF;

	//
//	IF 6=uMotorIndex THEN //ExtruderVisu
//		rData[0]	:= gExtruderB.ActSpeed;
//		rData[1]	:= gAcs380Ctrl.Status.ActCurrent[1]/100;
//		rData[2]	:= gAcs380Ctrl.Status.ActTorque[1]/100;
//		//	rData[3]	:= ;
//	END_IF;

	//----------------------------------
	//----------------------------------
	//Cursor
	Trace.Config.rCursorMove	:= Trace.Config.rHMICursorMove / 1000;
	//----------------------
	//Main
	CASE Trace.uStep OF
		0://INIT
			IF Trace.Cmd.bEnable THEN
				Trace.uDIndex	:= 0;
				Trace.uStep		:= 20;
				memset(ADR(Trace.Data),0,SIZEOF(Trace.Data)); //ipis0226
				//				FOR Trace.uTraceIndex := 0 TO MAX_NUM DO
				//
//				END_FOR;
			END_IF;
		20://Data -> Trend
			IF Trace.uDIndex < MAX_DATA THEN
				FOR Trace.uTraceIndex := 0 TO MAX_NUM DO
					Trace.Data[Trace.uTraceIndex].rData[Trace.uDIndex]	:= rData[Trace.uTraceIndex];
					//YMax
					IF Trace.Data[Trace.uTraceIndex].rData[Trace.uDIndex] >= Trace.Data[Trace.uTraceIndex].rYDMax THEN
						Trace.Data[Trace.uTraceIndex].rYMax := Trace.Data[Trace.uTraceIndex].rData[Trace.uDIndex] * 1.1;
						Trace.Data[Trace.uTraceIndex].rYDMax := Trace.Data[Trace.uTraceIndex].rData[Trace.uDIndex];
					END_IF;
					//YMin
					IF Trace.Data[Trace.uTraceIndex].rData[Trace.uDIndex] <= Trace.Data[Trace.uTraceIndex].rYDMin THEN
						Trace.Data[Trace.uTraceIndex].rYMin := Trace.Data[Trace.uTraceIndex].rData[Trace.uDIndex] * 1.1;
						Trace.Data[Trace.uTraceIndex].rYDMin := Trace.Data[Trace.uTraceIndex].rData[Trace.uDIndex];
					END_IF;
				END_FOR;
				Trace.uDIndex := Trace.uDIndex + 1;
			ELSE
				Trace.Cmd.bEnable	:= FALSE;
				Trace.uStep			:= 0;
			END_IF;
	END_CASE;
	//----------------------
END_PROGRAM
```

#### Init.st - Init code
```iecst
PROGRAM _INIT
	(* Insert code here *)
	Trace.uDIndex := MAX_DATA;  // VC4 trend bug for cursor

	(******Trend Option******)
	memset(ADR(uOptMotionTrend), 2, SIZEOF(uOptMotionTrend));
	uOptMotionTrend[0]  	:= 0;//RClamp
//	uOptMotionTrend[1]  	:= 0;//LClamp
	uOptMotionTrend[2]  	:= 0;//RCarriage
//	uOptMotionTrend[3]  	:= 0;//LCarriage
	uOptMotionTrend[4]  	:= 0;//RBlowpin1
//	uOptMotionTrend[5]  	:= 0;//LBlowpin1
	uOptMotionTrend[6]  	:= 0;//RRobotTransfer
//	uOptMotionTrend[7]  	:= 0;//LRobotTransfer
	uOptMotionTrend[10]  	:= 0;//Extrlift
	uOptMotionTrend[11]  	:= 0;//Parison
//	uOptMotionTrend[14]  	:= 0;//RBlowpin2
	//	uOptMotionTrend[15]  	:= 0;//LBlowpin2

	//Max Torque Set
	gMotorTrace.RMold.Clamp.Max_Torque_Set := 104;
	gMotorTrace.RMold.Carriage.Max_Torque_Set := 31;
	gMotorTrace.RMold.BlowPin.Max_Torque_Set := 38.7;
	gMotorTrace.Extrlift.Max_Torque_Set := 3.3;
	gMotorTrace.Parison.Max_Torque_Set := 12.6;

END_PROGRAM
```

#### Types.typ - Local data types
```iecst
(*Insert your comment here.*)

TYPE
	TraceData_typ : 	STRUCT
		rData : ARRAY[0..MAX_DATA]OF REAL;
		rYDMin : REAL; (*實際最小值*)
		rYDMax : REAL; (*實際最大值*)
		rYMin : REAL; (*人機顯示最小值，目的為了讓曲線更集中*)
		rYMax : REAL; (*人機顯示最大值，目的為了讓曲線更集中*)
		rCursorX : REAL; (*第幾筆資料*)
		rCursorY : REAL; (*光標資料*)
	END_STRUCT;
	TraceConfig_typ : 	STRUCT
		rZoomX : REAL;
		rScrollX : REAL;
		rCursorMove : REAL;
		rHMICursorMove : REAL; (*重疊在Trend上元件，目的是為了直接點圖找位置*)
	END_STRUCT;
	TraceCmd_typ : 	STRUCT
		bEnable : BOOL; (*啟動後，開始擷取資料，擷取完畢，自動清為0*)
		bHideY : USINT;
		bHideX : USINT;
		bHideData : ARRAY[0..MAX_NUM]OF USINT;
	END_STRUCT;
	Trace_typ : 	STRUCT
		uStep : UINT;
		uTraceIndex : UINT; (*Channel Index*)
		uDIndex : UINT; (*資料Index*)
		Data : ARRAY[0..MAX_NUM]OF TraceData_typ;
		Config : TraceConfig_typ;
		Cmd : TraceCmd_typ;
	END_STRUCT;
END_TYPE
```
